LIN {X 0,Y 474.698,Z 275.654,A -85,B 0,C 180,E1 -7395.456,E2 -7395.456} C_VEL
LIN {X 0,Y 474.663,Z 275.673,A -85,B 0,C 180,E1 -7399.01,E2 -7399.01} C_VEL
LIN {X 0,Y 474.587,Z 275.663,A -85,B 0,C 180,E1 -7401.729,E2 -7401.729} C_VEL
LIN {X 0,Y 474.657,Z 275.67,A -85,B 0,C 180,E1 -7404.493,E2 -7404.493} C_VEL
LIN {X 0,Y 474.679,Z 275.656,A -85,B 0,C 180,E1 -7407.335,E2 -7407.335} C_VEL
LIN {X 0,Y 474.603,Z 275.676,A -85,B 0,C 180,E1 -7410.23,E2 -7410.23} C_VEL
LIN {X 0,Y 474.641,Z 275.673,A -85,B 0,C 180,E1 -7413.22,E2 -7413.22} C_VEL
LIN {X 0,Y 474.592,Z 275.678,A -85,B 0,C 180,E1 -7416.323,E2 -7416.323} C_VEL
LIN {X 0,Y 474.616,Z 275.673,A -85,B 0,C 180,E1 -7419.646,E2 -7419.646} C_VEL
LIN {X 0,Y 474.63,Z 275.671,A -85,B 0,C 180,E1 -7422.933,E2 -7422.933} C_VEL
LIN {X 0,Y 474.608,Z 275.668,A -85,B 0,C 180,E1 -7425.895,E2 -7425.895} C_VEL
LIN {X 0,Y 474.627,Z 275.678,A -85,B 0,C 180,E1 -7429.041,E2 -7429.041} C_VEL
LIN {X 0,Y 474.609,Z 275.671,A -85,B 0,C 180,E1 -7431.704,E2 -7431.704} C_VEL
LIN {X 0,Y 474.624,Z 275.678,A -85,B 0,C 180,E1 -7434.726,E2 -7434.726} C_VEL
LIN {X 0,Y 474.635,Z 275.669,A -85,B 0,C 180,E1 -7437.788,E2 -7437.788} C_VEL
LIN {X 0,Y 474.657,Z 275.717,A -85,B 0,C 180,E1 -7439.725,E2 -7439.725} C_VEL
LIN {X 0,Y 477.611,Z 285.664,A -85,B 0,C 180,E1 -7441.163,E2 -7441.163} C_VEL
LIN {X 0,Y 486.377,Z 304.406,A -85,B 0,C 180,E1 -7442.044,E2 -7442.044} C_VEL
LIN {X 0,Y 486.586,Z 308.524,A -85,B 0,C 180,E1 -7442.124,E2 -7442.124} C_VEL
LIN {X 0,Y 485.977,Z 352.152,A -85,B 0,C 180,E1 -7442.8,E2 -7442.8} C_VEL
LIN {X 0,Y 485.357,Z 358.003,A -85,B 0,C 180,E1 -7442.857,E2 -7442.857} C_VEL
LIN {X 0,Y 479.946,Z 377.102,A -85,B 0,C 180,E1 -7442.838,E2 -7442.838} C_VEL
LIN {X 0,Y 479.226,Z 382.961,A -85,B 0,C 180,E1 -7442.89,E2 -7442.89} C_VEL
LIN {X 0,Y 477.794,Z 488.089,A -85,B 0,C 180,E1 -7444.548,E2 -7444.548} C_VEL
LIN {X 0,Y 477.341,Z 503.327,A -85,B 0,C 180,E1 -7444.899,E2 -7444.899} C_VEL
LIN {X 0,Y 476.655,Z 519.69,A -85,B 0,C 180,E1 -7445.443,E2 -7445.443} C_VEL
LIN {X 0,Y 475.799,Z 535.126,A -85,B 0,C 180,E1 -7446.132,E2 -7446.132} C_VEL
LIN {X 0,Y 474.828,Z 550.129,A -85,B 0,C 180,E1 -7446.975,E2 -7446.975} C_VEL
LIN {X 0,Y 473.716,Z 565.062,A -85,B 0,C 180,E1 -7448,E2 -7448} C_VEL
LIN {X 0,Y 472.635,Z 578.371,A -85,B 0,C 180,E1 -7449.092,E2 -7449.092} C_VEL
LIN {X 0,Y 471.51,Z 591.755,A -85,B 0,C 180,E1 -7450.405,E2 -7450.405} C_VEL
LIN {X 0,Y 470.479,Z 603.142,A -85,B 0,C 180,E1 -7451.718,E2 -7451.718} C_VEL
LIN {X 0,Y 469.522,Z 615.062,A -85,B 0,C 180,E1 -7453.331,E2 -7453.331} C_VEL
LIN {X 0,Y 468.699,Z 625.549,A -85,B 0,C 180,E1 -7455.01,E2 -7455.01} C_VEL
LIN {X 0,Y 467.993,Z 634.788,A -85,B 0,C 180,E1 -7456.761,E2 -7456.761} C_VEL
LIN {X 0,Y 467.476,Z 643.328,A -85,B 0,C 180,E1 -7458.73,E2 -7458.73} C_VEL
LIN {X 0,Y 467.036,Z 650.904,A -85,B 0,C 180,E1 -7460.909,E2 -7460.909} C_VEL
LIN {X 0,Y 466.857,Z 655.603,A -85,B 0,C 180,E1 -7462.648,E2 -7462.648} C_VEL
LIN {X 0,Y 466.786,Z 658.459,A -85,B 0,C 180,E1 -7463.95,E2 -7463.95} C_VEL
LIN {X 0,Y 466.637,Z 661.374,A -85,B 0,C 180,E1 -7465.681,E2 -7465.681} C_VEL
LIN {X 0,Y 466.674,Z 663.284,A -85,B 0,C 180,E1 -7467.411,E2 -7467.411} C_VEL
LIN {X 0,Y 466.616,Z 664.26,A -85,B 0,C 180,E1 -7469.137,E2 -7469.137} C_VEL
LIN {X 0,Y 466.615,Z 664.276,A -85,B 0,C 180,E1 -7470.863,E2 -7470.863} C_VEL
LIN {X 0,Y 466.674,Z 663.368,A -85,B 0,C 180,E1 -7472.589,E2 -7472.589} C_VEL
LIN {X 0,Y 466.636,Z 661.491,A -85,B 0,C 180,E1 -7474.319,E2 -7474.319} C_VEL
LIN {X 0,Y 466.808,Z 657.814,A -85,B 0,C 180,E1 -7476.456,E2 -7476.456} C_VEL
LIN {X 0,Y 466.958,Z 653.633,A -85,B 0,C 180,E1 -7478.22,E2 -7478.22} C_VEL
LIN {X 0,Y 467.131,Z 648.378,A -85,B 0,C 180,E1 -7479.963,E2 -7479.963} C_VEL
LIN {X 0,Y 467.549,Z 641.906,A -85,B 0,C 180,E1 -7481.708,E2 -7481.708} C_VEL
LIN {X 0,Y 468.046,Z 634.141,A -85,B 0,C 180,E1 -7483.458,E2 -7483.458} C_VEL
LIN {X 0,Y 468.755,Z 624.825,A -85,B 0,C 180,E1 -7485.211,E2 -7485.211} C_VEL
LIN {X 0,Y 469.626,Z 613.968,A -85,B 0,C 180,E1 -7486.922,E2 -7486.922} C_VEL
LIN {X 0,Y 470.594,Z 602.088,A -85,B 0,C 180,E1 -7488.503,E2 -7488.503} C_VEL
LIN {X 0,Y 471.667,Z 589.425,A -85,B 0,C 180,E1 -7489.928,E2 -7489.928} C_VEL
LIN {X 0,Y 472.899,Z 575.579,A -85,B 0,C 180,E1 -7491.238,E2 -7491.238} C_VEL
LIN {X 0,Y 473.973,Z 561.898,A -85,B 0,C 180,E1 -7492.331,E2 -7492.331} C_VEL
LIN {X 0,Y 475.059,Z 546.493,A -85,B 0,C 180,E1 -7493.344,E2 -7493.344} C_VEL
LIN {X 0,Y 475.946,Z 531.63,A -85,B 0,C 180,E1 -7494.132,E2 -7494.132} C_VEL
LIN {X 0,Y 476.877,Z 515.29,A -85,B 0,C 180,E1 -7494.807,E2 -7494.807} C_VEL
LIN {X 0,Y 477.391,Z 500.575,A -85,B 0,C 180,E1 -7495.273,E2 -7495.273} C_VEL
LIN {X 0,Y 477.922,Z 482.833,A -85,B 0,C 180,E1 -7495.638,E2 -7495.638} C_VEL
LIN {X 0,Y 480.341,Z 306.951,A -85,B 0,C 180,E1 -7498.393,E2 -7498.393} C_VEL
LIN {X 0,Y 470.381,Z 285.74,A -85,B 0,C 180,E1 -7499.424,E2 -7499.424} C_VEL
LIN {X 0,Y 467.558,Z 276.56,A -85,B 0,C 180,E1 -7500.82,E2 -7500.82} C_VEL
LIN {X 0,Y 467.585,Z 276.553,A -85,B 0,C 180,E1 -7503.788,E2 -7503.788} C_VEL
LIN {X 0,Y 467.541,Z 276.547,A -85,B 0,C 180,E1 -7507.185,E2 -7507.185} C_VEL
LIN {X 0,Y 467.573,Z 276.551,A -85,B 0,C 180,E1 -7510.265,E2 -7510.265} C_VEL
LIN {X 0,Y 467.585,Z 276.548,A -85,B 0,C 180,E1 -7512.567,E2 -7512.567} C_VEL
LIN {X 0,Y 467.569,Z 276.553,A -85,B 0,C 180,E1 -7515.053,E2 -7515.053} C_VEL
LIN {X 0,Y 467.587,Z 276.553,A -85,B 0,C 180,E1 -7517.44,E2 -7517.44} C_VEL
LIN {X 0,Y 467.574,Z 276.554,A -85,B 0,C 180,E1 -7520.854,E2 -7520.854} C_VEL
LIN {X 0,Y 467.56,Z 276.552,A -85,B 0,C 180,E1 -7524.26,E2 -7524.26} C_VEL
LIN {X 0,Y 467.579,Z 276.547,A -85,B 0,C 180,E1 -7527.321,E2 -7527.321} C_VEL
LIN {X 0,Y 467.568,Z 276.554,A -85,B 0,C 180,E1 -7530.667,E2 -7530.667} C_VEL
LIN {X 0,Y 467.614,Z 276.543,A -85,B 0,C 180,E1 -7533.199,E2 -7533.199} C_VEL
LIN {X 0,Y 467.591,Z 276.548,A -85,B 0,C 180,E1 -7536.468,E2 -7536.468} C_VEL
LIN {X 0,Y 467.62,Z 276.545,A -85,B 0,C 180,E1 -7539.777,E2 -7539.777} C_VEL
LIN {X 0,Y 467.604,Z 276.547,A -85,B 0,C 180,E1 -7542.506,E2 -7542.506} C_VEL
LIN {X 0,Y 467.604,Z 276.544,A -85,B 0,C 180,E1 -7545.196,E2 -7545.196} C_VEL
LIN {X 0,Y 467.653,Z 276.54,A -85,B 0,C 180,E1 -7547.854,E2 -7547.854} C_VEL
LIN {X 0,Y 467.677,Z 276.534,A -85,B 0,C 180,E1 -7551.357,E2 -7551.357} C_VEL
LIN {X 0,Y 467.743,Z 276.53,A -85,B 0,C 180,E1 -7553.962,E2 -7553.962} C_VEL
LIN {X 0,Y 467.857,Z 276.506,A -85,B 0,C 180,E1 -7557.417,E2 -7557.417} C_VEL
LIN {X 0,Y 467.88,Z 276.512,A -85,B 0,C 180,E1 -7560,E2 -7560} C_VEL
LIN {X 0,Y 467.857,Z 276.516,A -85,B 0,C 180,E1 -7562.583,E2 -7562.583} C_VEL
LIN {X 0,Y 467.742,Z 276.527,A -85,B 0,C 180,E1 -7566.037,E2 -7566.037} C_VEL
LIN {X 0,Y 467.678,Z 276.542,A -85,B 0,C 180,E1 -7568.643,E2 -7568.643} C_VEL
LIN {X 0,Y 467.653,Z 276.537,A -85,B 0,C 180,E1 -7572.145,E2 -7572.145} C_VEL
LIN {X 0,Y 467.636,Z 276.543,A -85,B 0,C 180,E1 -7575.695,E2 -7575.695} C_VEL
LIN {X 0,Y 467.614,Z 276.549,A -85,B 0,C 180,E1 -7578.765,E2 -7578.765} C_VEL
LIN {X 0,Y 467.577,Z 276.553,A -85,B 0,C 180,E1 -7581.268,E2 -7581.268} C_VEL
LIN {X 0,Y 467.57,Z 276.552,A -85,B 0,C 180,E1 -7583.943,E2 -7583.943} C_VEL
LIN {X 0,Y 467.613,Z 276.553,A -85,B 0,C 180,E1 -7586.8,E2 -7586.8} C_VEL
LIN {X 0,Y 467.551,Z 276.555,A -85,B 0,C 180,E1 -7589.738,E2 -7589.738} C_VEL
LIN {X 0,Y 467.58,Z 276.557,A -85,B 0,C 180,E1 -7592.758,E2 -7592.758} C_VEL
LIN {X 0,Y 467.554,Z 276.554,A -85,B 0,C 180,E1 -7595.889,E2 -7595.889} C_VEL
LIN {X 0,Y 467.579,Z 276.557,A -85,B 0,C 180,E1 -7599.145,E2 -7599.145} C_VEL
LIN {X 0,Y 467.583,Z 276.558,A -85,B 0,C 180,E1 -7602.567,E2 -7602.567} C_VEL
LIN {X 0,Y 467.568,Z 276.559,A -85,B 0,C 180,E1 -7605.053,E2 -7605.053} C_VEL
LIN {X 0,Y 467.586,Z 276.553,A -85,B 0,C 180,E1 -7607.44,E2 -7607.44} C_VEL
LIN {X 0,Y 467.579,Z 276.557,A -85,B 0,C 180,E1 -7610.855,E2 -7610.855} C_VEL
LIN {X 0,Y 467.557,Z 276.559,A -85,B 0,C 180,E1 -7614.261,E2 -7614.261} C_VEL
LIN {X 0,Y 467.618,Z 276.563,A -85,B 0,C 180,E1 -7616.732,E2 -7616.732} C_VEL
LIN {X 0,Y 473.316,Z 295.045,A -85,B 0,C 180,E1 -7619.243,E2 -7619.243} C_VEL
LIN {X 0,Y 475.745,Z 303.396,A -85,B 0,C 180,E1 -7620.329,E2 -7620.329} C_VEL
LIN {X 0,Y 475.862,Z 305.952,A -85,B 0,C 180,E1 -7620.618,E2 -7620.618} C_VEL
LIN {X 0,Y 475.685,Z 309.709,A -85,B 0,C 180,E1 -7620.982,E2 -7620.982} C_VEL
LIN {X 0,Y 480.083,Z 335.198,A -85,B 0,C 180,E1 -7621.695,E2 -7621.695} C_VEL
LIN {X 0,Y 477.574,Z 515.045,A -85,B 0,C 180,E1 -7624.523,E2 -7624.523} C_VEL
LIN {X 0,Y 476.934,Z 530.938,A -85,B 0,C 180,E1 -7624.906,E2 -7624.906} C_VEL
LIN {X 0,Y 476.204,Z 547.344,A -85,B 0,C 180,E1 -7625.476,E2 -7625.476} C_VEL
LIN {X 0,Y 475.296,Z 561.77,A -85,B 0,C 180,E1 -7626.123,E2 -7626.123} C_VEL
LIN {X 0,Y 474.374,Z 576.069,A -85,B 0,C 180,E1 -7626.934,E2 -7626.934} C_VEL
LIN {X 0,Y 473.143,Z 591.267,A -85,B 0,C 180,E1 -7627.972,E2 -7627.972} C_VEL
LIN {X 0,Y 471.982,Z 605.787,A -85,B 0,C 180,E1 -7629.176,E2 -7629.176} C_VEL
LIN {X 0,Y 470.929,Z 618.532,A -85,B 0,C 180,E1 -7630.425,E2 -7630.425} C_VEL
LIN {X 0,Y 469.868,Z 631.368,A -85,B 0,C 180,E1 -7631.919,E2 -7631.919} C_VEL
LIN {X 0,Y 468.941,Z 643.342,A -85,B 0,C 180,E1 -7633.569,E2 -7633.569} C_VEL
LIN {X 0,Y 468.186,Z 653.464,A -85,B 0,C 180,E1 -7635.215,E2 -7635.215} C_VEL
LIN {X 0,Y 467.648,Z 662.611,A -85,B 0,C 180,E1 -7636.972,E2 -7636.972} C_VEL
LIN {X 0,Y 467.223,Z 670.275,A -85,B 0,C 180,E1 -7638.723,E2 -7638.723} C_VEL
LIN {X 0,Y 466.863,Z 677.966,A -85,B 0,C 180,E1 -7640.906,E2 -7640.906} C_VEL
LIN {X 0,Y 466.775,Z 682.744,A -85,B 0,C 180,E1 -7642.647,E2 -7642.647} C_VEL
LIN {X 0,Y 466.696,Z 685.653,A -85,B 0,C 180,E1 -7643.949,E2 -7643.949} C_VEL
LIN {X 0,Y 466.606,Z 688.604,A -85,B 0,C 180,E1 -7645.681,E2 -7645.681} C_VEL
LIN {X 0,Y 466.637,Z 690.549,A -85,B 0,C 180,E1 -7647.41,E2 -7647.41} C_VEL
LIN {X 0,Y 466.614,Z 691.513,A -85,B 0,C 180,E1 -7649.137,E2 -7649.137} C_VEL
LIN {X 0,Y 466.614,Z 691.512,A -85,B 0,C 180,E1 -7650.863,E2 -7650.863} C_VEL
LIN {X 0,Y 466.637,Z 690.548,A -85,B 0,C 180,E1 -7652.59,E2 -7652.59} C_VEL
LIN {X 0,Y 466.606,Z 688.603,A -85,B 0,C 180,E1 -7654.319,E2 -7654.319} C_VEL
LIN {X 0,Y 466.748,Z 684.941,A -85,B 0,C 180,E1 -7656.393,E2 -7656.393} C_VEL
LIN {X 0,Y 466.834,Z 680.493,A -85,B 0,C 180,E1 -7658.223,E2 -7658.223} C_VEL
LIN {X 0,Y 466.981,Z 675.097,A -85,B 0,C 180,E1 -7659.967,E2 -7659.967} C_VEL
LIN {X 0,Y 467.36,Z 668.451,A -85,B 0,C 180,E1 -7661.713,E2 -7661.713} C_VEL
LIN {X 0,Y 467.749,Z 660.487,A -85,B 0,C 180,E1 -7663.467,E2 -7663.467} C_VEL
LIN {X 0,Y 468.449,Z 650.979,A -85,B 0,C 180,E1 -7665.221,E2 -7665.221} C_VEL
LIN {X 0,Y 469.272,Z 639.594,A -85,B 0,C 180,E1 -7666.98,E2 -7666.98} C_VEL
LIN {X 0,Y 470.247,Z 627.776,A -85,B 0,C 180,E1 -7668.517,E2 -7668.517} C_VEL
LIN {X 0,Y 471.239,Z 615.474,A -85,B 0,C 180,E1 -7669.884,E2 -7669.884} C_VEL
LIN {X 0,Y 472.283,Z 602.081,A -85,B 0,C 180,E1 -7671.153,E2 -7671.153} C_VEL
LIN {X 0,Y 473.375,Z 588.383,A -85,B 0,C 180,E1 -7672.246,E2 -7672.246} C_VEL
LIN {X 0,Y 474.499,Z 573.377,A -85,B 0,C 180,E1 -7673.233,E2 -7673.233} C_VEL
LIN {X 0,Y 475.517,Z 558.339,A -85,B 0,C 180,E1 -7674.039,E2 -7674.039} C_VEL
LIN {X 0,Y 476.42,Z 542.396,A -85,B 0,C 180,E1 -7674.716,E2 -7674.716} C_VEL
LIN {X 0,Y 477.177,Z 526.233,A -85,B 0,C 180,E1 -7675.226,E2 -7675.226} C_VEL
LIN {X 0,Y 477.681,Z 509.478,A -85,B 0,C 180,E1 -7675.577,E2 -7675.577} C_VEL
LIN {X 0,Y 480.11,Z 334.584,A -85,B 0,C 180,E1 -7678.312,E2 -7678.312} C_VEL
LIN {X 0,Y 475.615,Z 309.029,A -85,B 0,C 180,E1 -7679.057,E2 -7679.057} C_VEL
LIN {X 0,Y 475.783,Z 303.384,A -85,B 0,C 180,E1 -7679.666,E2 -7679.666} C_VEL
LIN {X 0,Y 470.106,Z 284.516,A -85,B 0,C 180,E1 -7682.165,E2 -7682.165} C_VEL
LIN {X 0,Y 467.619,Z 276.543,A -85,B 0,C 180,E1 -7683.268,E2 -7683.268} C_VEL
LIN {X 0,Y 467.551,Z 276.558,A -85,B 0,C 180,E1 -7685.89,E2 -7685.89} C_VEL
LIN {X 0,Y 467.58,Z 276.555,A -85,B 0,C 180,E1 -7689.145,E2 -7689.145} C_VEL
LIN {X 0,Y 467.584,Z 276.551,A -85,B 0,C 180,E1 -7692.567,E2 -7692.567} C_VEL
LIN {X 0,Y 467.568,Z 276.554,A -85,B 0,C 180,E1 -7695.053,E2 -7695.053} C_VEL
LIN {X 0,Y 467.586,Z 276.551,A -85,B 0,C 180,E1 -7697.44,E2 -7697.44} C_VEL
LIN {X 0,Y 467.573,Z 276.55,A -85,B 0,C 180,E1 -7700.855,E2 -7700.855} C_VEL
LIN {X 0,Y 467.559,Z 276.551,A -85,B 0,C 180,E1 -7704.26,E2 -7704.26} C_VEL
LIN {X 0,Y 467.579,Z 276.553,A -85,B 0,C 180,E1 -7707.321,E2 -7707.321} C_VEL
LIN {X 0,Y 467.567,Z 276.551,A -85,B 0,C 180,E1 -7710.667,E2 -7710.667} C_VEL
LIN {X 0,Y 467.614,Z 276.55,A -85,B 0,C 180,E1 -7713.2,E2 -7713.2} C_VEL
LIN {X 0,Y 467.59,Z 276.549,A -85,B 0,C 180,E1 -7716.468,E2 -7716.468} C_VEL
LIN {X 0,Y 467.62,Z 276.532,A -85,B 0,C 180,E1 -7719.777,E2 -7719.777} C_VEL
LIN {X 0,Y 467.604,Z 276.547,A -85,B 0,C 180,E1 -7722.507,E2 -7722.507} C_VEL
LIN {X 0,Y 467.603,Z 276.541,A -85,B 0,C 180,E1 -7725.197,E2 -7725.197} C_VEL
LIN {X 0,Y 467.653,Z 276.536,A -85,B 0,C 180,E1 -7727.855,E2 -7727.855} C_VEL
LIN {X 0,Y 467.679,Z 276.536,A -85,B 0,C 180,E1 -7731.357,E2 -7731.357} C_VEL
LIN {X 0,Y 467.743,Z 276.516,A -85,B 0,C 180,E1 -7733.963,E2 -7733.963} C_VEL
LIN {X 0,Y 467.857,Z 276.518,A -85,B 0,C 180,E1 -7737.417,E2 -7737.417} C_VEL
LIN {X 0,Y 467.88,Z 276.501,A -85,B 0,C 180,E1 -7740,E2 -7740} C_VEL
LIN {X 0,Y 467.858,Z 276.509,A -85,B 0,C 180,E1 -7742.583,E2 -7742.583} C_VEL
LIN {X 0,Y 467.733,Z 276.528,A -85,B 0,C 180,E1 -7746.038,E2 -7746.038} C_VEL
LIN {X 0,Y 467.679,Z 276.523,A -85,B 0,C 180,E1 -7748.643,E2 -7748.643} C_VEL
LIN {X 0,Y 467.654,Z 276.541,A -85,B 0,C 180,E1 -7752.146,E2 -7752.146} C_VEL
LIN {X 0,Y 467.637,Z 276.533,A -85,B 0,C 180,E1 -7755.695,E2 -7755.695} C_VEL
LIN {X 0,Y 467.615,Z 276.551,A -85,B 0,C 180,E1 -7758.765,E2 -7758.765} C_VEL
LIN {X 0,Y 467.578,Z 276.539,A -85,B 0,C 180,E1 -7761.268,E2 -7761.268} C_VEL
LIN {X 0,Y 467.571,Z 276.55,A -85,B 0,C 180,E1 -7763.943,E2 -7763.943} C_VEL
LIN {X 0,Y 467.615,Z 276.543,A -85,B 0,C 180,E1 -7766.8,E2 -7766.8} C_VEL
LIN {X 0,Y 467.552,Z 276.553,A -85,B 0,C 180,E1 -7769.738,E2 -7769.738} C_VEL
LIN {X 0,Y 467.582,Z 276.553,A -85,B 0,C 180,E1 -7772.759,E2 -7772.759} C_VEL
LIN {X 0,Y 467.555,Z 276.552,A -85,B 0,C 180,E1 -7775.89,E2 -7775.89} C_VEL
LIN {X 0,Y 467.574,Z 276.551,A -85,B 0,C 180,E1 -7779.146,E2 -7779.146} C_VEL
LIN {X 0,Y 467.585,Z 276.545,A -85,B 0,C 180,E1 -7782.567,E2 -7782.567} C_VEL
LIN {X 0,Y 467.569,Z 276.55,A -85,B 0,C 180,E1 -7785.053,E2 -7785.053} C_VEL
LIN {X 0,Y 467.588,Z 276.552,A -85,B 0,C 180,E1 -7787.44,E2 -7787.44} C_VEL
LIN {X 0,Y 467.582,Z 276.554,A -85,B 0,C 180,E1 -7790.856,E2 -7790.856} C_VEL
LIN {X 0,Y 467.559,Z 276.552,A -85,B 0,C 180,E1 -7794.261,E2 -7794.261} C_VEL
LIN {X 0,Y 467.581,Z 276.542,A -85,B 0,C 180,E1 -7797.321,E2 -7797.321} C_VEL
LIN {X 0,Y 467.581,Z 276.568,A -85,B 0,C 180,E1 -7799.299,E2 -7799.299} C_VEL
LIN {X 0,Y 470.498,Z 286.066,A -85,B 0,C 180,E1 -7800.687,E2 -7800.687} C_VEL
LIN {X 0,Y 480.235,Z 306.732,A -85,B 0,C 180,E1 -7801.689,E2 -7801.689} C_VEL
LIN {X 0,Y 479.226,Z 382.961,A -85,B 0,C 180,E1 -7802.89,E2 -7802.89} C_VEL
LIN {X 0,Y 478.525,Z 388.81,A -85,B 0,C 180,E1 -7802.944,E2 -7802.944} C_VEL
LIN {X 0,Y 473.174,Z 407.9,A -85,B 0,C 180,E1 -7802.929,E2 -7802.929} C_VEL
LIN {X 0,Y 472.476,Z 413.75,A -85,B 0,C 180,E1 -7802.983,E2 -7802.983} C_VEL
LIN {X 0,Y 471.384,Z 488.455,A -85,B 0,C 180,E1 -7804.179,E2 -7804.179} C_VEL
LIN {X 0,Y 470.848,Z 505.377,A -85,B 0,C 180,E1 -7804.588,E2 -7804.588} C_VEL
LIN {X 0,Y 470.137,Z 521.212,A -85,B 0,C 180,E1 -7805.138,E2 -7805.138} C_VEL
LIN {X 0,Y 469.272,Z 536.355,A -85,B 0,C 180,E1 -7805.832,E2 -7805.832} C_VEL
LIN {X 0,Y 468.266,Z 550.66,A -85,B 0,C 180,E1 -7806.654,E2 -7806.654} C_VEL
LIN {X 0,Y 467.129,Z 565.276,A -85,B 0,C 180,E1 -7807.673,E2 -7807.673} C_VEL
LIN {X 0,Y 465.997,Z 578.584,A -85,B 0,C 180,E1 -7808.78,E2 -7808.78} C_VEL
LIN {X 0,Y 464.759,Z 591.969,A -85,B 0,C 180,E1 -7810.109,E2 -7810.109} C_VEL
LIN {X 0,Y 463.682,Z 603.355,A -85,B 0,C 180,E1 -7811.44,E2 -7811.44} C_VEL
LIN {X 0,Y 462.696,Z 614.91,A -85,B 0,C 180,E1 -7813.022,E2 -7813.022} C_VEL
LIN {X 0,Y 461.883,Z 624.527,A -85,B 0,C 180,E1 -7814.557,E2 -7814.557} C_VEL
LIN {X 0,Y 461.101,Z 633.901,A -85,B 0,C 180,E1 -7816.335,E2 -7816.335} C_VEL
LIN {X 0,Y 460.558,Z 641.75,A -85,B 0,C 180,E1 -7818.112,E2 -7818.112} C_VEL
LIN {X 0,Y 460.096,Z 648.3,A -85,B 0,C 180,E1 -7819.883,E2 -7819.883} C_VEL
LIN {X 0,Y 459.895,Z 653.592,A -85,B 0,C 180,E1 -7821.653,E2 -7821.653} C_VEL
LIN {X 0,Y 459.717,Z 658.082,A -85,B 0,C 180,E1 -7823.564,E2 -7823.564} C_VEL
LIN {X 0,Y 459.553,Z 661.583,A -85,B 0,C 180,E1 -7825.615,E2 -7825.615} C_VEL
LIN {X 0,Y 459.596,Z 663.492,A -85,B 0,C 180,E1 -7827.371,E2 -7827.371} C_VEL
LIN {X 0,Y 459.519,Z 664.467,A -85,B 0,C 180,E1 -7829.124,E2 -7829.124} C_VEL
LIN {X 0,Y 459.519,Z 664.483,A -85,B 0,C 180,E1 -7830.876,E2 -7830.876} C_VEL
LIN {X 0,Y 459.596,Z 663.574,A -85,B 0,C 180,E1 -7832.629,E2 -7832.629} C_VEL
LIN {X 0,Y 459.552,Z 661.698,A -85,B 0,C 180,E1 -7834.385,E2 -7834.385} C_VEL
LIN {X 0,Y 459.717,Z 658.262,A -85,B 0,C 180,E1 -7836.435,E2 -7836.435} C_VEL
LIN {X 0,Y 459.891,Z 653.839,A -85,B 0,C 180,E1 -7838.347,E2 -7838.347} C_VEL
LIN {X 0,Y 460.079,Z 648.585,A -85,B 0,C 180,E1 -7840.118,E2 -7840.118} C_VEL
LIN {X 0,Y 460.528,Z 642.113,A -85,B 0,C 180,E1 -7841.889,E2 -7841.889} C_VEL
LIN {X 0,Y 461.083,Z 634.348,A -85,B 0,C 180,E1 -7843.666,E2 -7843.666} C_VEL
LIN {X 0,Y 461.847,Z 625.032,A -85,B 0,C 180,E1 -7845.444,E2 -7845.444} C_VEL
LIN {X 0,Y 462.766,Z 614.174,A -85,B 0,C 180,E1 -7847.18,E2 -7847.18} C_VEL
LIN {X 0,Y 463.837,Z 602.292,A -85,B 0,C 180,E1 -7848.782,E2 -7848.782} C_VEL
LIN {X 0,Y 464.936,Z 589.63,A -85,B 0,C 180,E1 -7850.229,E2 -7850.229} C_VEL
LIN {X 0,Y 466.16,Z 577.067,A -85,B 0,C 180,E1 -7851.444,E2 -7851.444} C_VEL
LIN {X 0,Y 467.279,Z 563.561,A -85,B 0,C 180,E1 -7852.552,E2 -7852.552} C_VEL
LIN {X 0,Y 468.373,Z 549.154,A -85,B 0,C 180,E1 -7853.533,E2 -7853.533} C_VEL
LIN {X 0,Y 469.399,Z 532.954,A -85,B 0,C 180,E1 -7854.432,E2 -7854.432} C_VEL
LIN {X 0,Y 470.405,Z 516.245,A -85,B 0,C 180,E1 -7855.142,E2 -7855.142} C_VEL
LIN {X 0,Y 470.982,Z 500.763,A -85,B 0,C 180,E1 -7855.641,E2 -7855.641} C_VEL
LIN {X 0,Y 471.538,Z 483.554,A -85,B 0,C 180,E1 -7856.001,E2 -7856.001} C_VEL
LIN {X 0,Y 474.061,Z 308.964,A -85,B 0,C 180,E1 -7858.773,E2 -7858.773} C_VEL
LIN {X 0,Y 464.278,Z 288.306,A -85,B 0,C 180,E1 -7859.804,E2 -7859.804} C_VEL
LIN {X 0,Y 463.104,Z 285.806,A -85,B 0,C 180,E1 -7859.954,E2 -7859.954} C_VEL
LIN {X 0,Y 460.536,Z 277.44,A -85,B 0,C 180,E1 -7861.255,E2 -7861.255} C_VEL
LIN {X 0,Y 460.53,Z 277.435,A -85,B 0,C 180,E1 -7864.505,E2 -7864.505} C_VEL
LIN {X 0,Y 460.497,Z 277.43,A -85,B 0,C 180,E1 -7867.623,E2 -7867.623} C_VEL
LIN {X 0,Y 460.538,Z 277.427,A -85,B 0,C 180,E1 -7870.269,E2 -7870.269} C_VEL
LIN {X 0,Y 460.499,Z 277.436,A -85,B 0,C 180,E1 -7873.375,E2 -7873.375} C_VEL
LIN {X 0,Y 460.498,Z 277.432,A -85,B 0,C 180,E1 -7876.624,E2 -7876.624} C_VEL
LIN {X 0,Y 460.537,Z 277.429,A -85,B 0,C 180,E1 -7879.731,E2 -7879.731} C_VEL
LIN {X 0,Y 460.498,Z 277.431,A -85,B 0,C 180,E1 -7882.523,E2 -7882.523} C_VEL
LIN {X 0,Y 460.546,Z 277.428,A -85,B 0,C 180,E1 -7885.624,E2 -7885.624} C_VEL
LIN {X 0,Y 460.535,Z 277.426,A -85,B 0,C 180,E1 -7888.744,E2 -7888.744} C_VEL
LIN {X 0,Y 460.579,Z 277.412,A -85,B 0,C 180,E1 -7892.254,E2 -7892.254} C_VEL
LIN {X 0,Y 460.557,Z 277.427,A -85,B 0,C 180,E1 -7894.705,E2 -7894.705} C_VEL
LIN {X 0,Y 460.508,Z 277.421,A -85,B 0,C 180,E1 -7897.571,E2 -7897.571} C_VEL
LIN {X 0,Y 460.566,Z 277.424,A -85,B 0,C 180,E1 -7900.384,E2 -7900.384} C_VEL
LIN {X 0,Y 460.561,Z 277.416,A -85,B 0,C 180,E1 -7903.146,E2 -7903.146} C_VEL
LIN {X 0,Y 460.552,Z 277.424,A -85,B 0,C 180,E1 -7905.868,E2 -7905.868} C_VEL
LIN {X 0,Y 460.607,Z 277.42,A -85,B 0,C 180,E1 -7908.559,E2 -7908.559} C_VEL
LIN {X 0,Y 460.692,Z 277.404,A -85,B 0,C 180,E1 -7912.108,E2 -7912.108} C_VEL
LIN {X 0,Y 460.696,Z 277.412,A -85,B 0,C 180,E1 -7914.748,E2 -7914.748} C_VEL
LIN {X 0,Y 460.798,Z 277.385,A -85,B 0,C 180,E1 -7917.377,E2 -7917.377} C_VEL
LIN {X 0,Y 460.851,Z 277.388,A -85,B 0,C 180,E1 -7920,E2 -7920} C_VEL
LIN {X 0,Y 460.822,Z 277.391,A -85,B 0,C 180,E1 -7922.622,E2 -7922.622} C_VEL
LIN {X 0,Y 460.708,Z 277.404,A -85,B 0,C 180,E1 -7926.13,E2 -7926.13} C_VEL
LIN {X 0,Y 460.625,Z 277.418,A -85,B 0,C 180,E1 -7928.776,E2 -7928.776} C_VEL
LIN {X 0,Y 460.61,Z 277.416,A -85,B 0,C 180,E1 -7932.445,E2 -7932.445} C_VEL
LIN {X 0,Y 460.597,Z 277.419,A -85,B 0,C 180,E1 -7935.997,E2 -7935.997} C_VEL
LIN {X 0,Y 460.568,Z 277.428,A -85,B 0,C 180,E1 -7938.902,E2 -7938.902} C_VEL
LIN {X 0,Y 460.512,Z 277.432,A -85,B 0,C 180,E1 -7941.486,E2 -7941.486} C_VEL
LIN {X 0,Y 460.539,Z 277.43,A -85,B 0,C 180,E1 -7944.332,E2 -7944.332} C_VEL
LIN {X 0,Y 460.57,Z 277.428,A -85,B 0,C 180,E1 -7947.244,E2 -7947.244} C_VEL
LIN {X 0,Y 460.507,Z 277.434,A -85,B 0,C 180,E1 -7950.24,E2 -7950.24} C_VEL
LIN {X 0,Y 460.526,Z 277.434,A -85,B 0,C 180,E1 -7953.325,E2 -7953.325} C_VEL
LIN {X 0,Y 460.476,Z 277.441,A -85,B 0,C 180,E1 -7956.529,E2 -7956.529} C_VEL
LIN {X 0,Y 460.542,Z 277.436,A -85,B 0,C 180,E1 -7958.898,E2 -7958.898} C_VEL
LIN {X 0,Y 460.52,Z 277.435,A -85,B 0,C 180,E1 -7962.181,E2 -7962.181} C_VEL
LIN {X 0,Y 460.517,Z 277.434,A -85,B 0,C 180,E1 -7965.412,E2 -7965.412} C_VEL
LIN {X 0,Y 460.532,Z 277.434,A -85,B 0,C 180,E1 -7968.397,E2 -7968.397} C_VEL
LIN {X 0,Y 460.524,Z 277.433,A -85,B 0,C 180,E1 -7971.267,E2 -7971.267} C_VEL
LIN {X 0,Y 460.507,Z 277.43,A -85,B 0,C 180,E1 -7974.554,E2 -7974.554} C_VEL
LIN {X 0,Y 460.574,Z 277.577,A -85,B 0,C 180,E1 -7976.301,E2 -7976.301} C_VEL
LIN {X 0,Y 466.451,Z 296.278,A -85,B 0,C 180,E1 -7978.905,E2 -7978.905} C_VEL
LIN {X 0,Y 469.323,Z 306.823,A -85,B 0,C 180,E1 -7980.288,E2 -7980.288} C_VEL
LIN {X 0,Y 469.173,Z 309.378,A -85,B 0,C 180,E1 -7980.537,E2 -7980.537} C_VEL
LIN {X 0,Y 473.809,Z 335.907,A -85,B 0,C 180,E1 -7981.3,E2 -7981.3} C_VEL
LIN {X 0,Y 471.346,Z 505.455,A -85,B 0,C 180,E1 -7983.984,E2 -7983.984} C_VEL
LIN {X 0,Y 470.837,Z 522.804,A -85,B 0,C 180,E1 -7984.324,E2 -7984.324} C_VEL
LIN {X 0,Y 470.064,Z 539.941,A -85,B 0,C 180,E1 -7984.839,E2 -7984.839} C_VEL
LIN {X 0,Y 469.151,Z 555.906,A -85,B 0,C 180,E1 -7985.496,E2 -7985.496} C_VEL
LIN {X 0,Y 468.238,Z 569.698,A -85,B 0,C 180,E1 -7986.215,E2 -7986.215} C_VEL
LIN {X 0,Y 467.032,Z 585.074,A -85,B 0,C 180,E1 -7987.202,E2 -7987.202} C_VEL
LIN {X 0,Y 465.867,Z 599.292,A -85,B 0,C 180,E1 -7988.309,E2 -7988.309} C_VEL
LIN {X 0,Y 464.717,Z 612.527,A -85,B 0,C 180,E1 -7989.53,E2 -7989.53} C_VEL
LIN {X 0,Y 463.671,Z 623.84,A -85,B 0,C 180,E1 -7990.751,E2 -7990.751} C_VEL
LIN {X 0,Y 462.615,Z 636.173,A -85,B 0,C 180,E1 -7992.312,E2 -7992.312} C_VEL
LIN {X 0,Y 461.756,Z 646.509,A -85,B 0,C 180,E1 -7993.843,E2 -7993.843} C_VEL
LIN {X 0,Y 461.057,Z 655.739,A -85,B 0,C 180,E1 -7995.433,E2 -7995.433} C_VEL
LIN {X 0,Y 460.531,Z 664.437,A -85,B 0,C 180,E1 -7997.216,E2 -7997.216} C_VEL
LIN {X 0,Y 460.102,Z 671.717,A -85,B 0,C 180,E1 -7998.993,E2 -7998.993} C_VEL
LIN {X 0,Y 459.787,Z 677.758,A -85,B 0,C 180,E1 -8000.764,E2 -8000.764} C_VEL
LIN {X 0,Y 459.648,Z 683.613,A -85,B 0,C 180,E1 -8002.974,E2 -8002.974} C_VEL
LIN {X 0,Y 459.578,Z 687.037,A -85,B 0,C 180,E1 -8004.736,E2 -8004.736} C_VEL
LIN {X 0,Y 459.56,Z 689.527,A -85,B 0,C 180,E1 -8006.493,E2 -8006.493} C_VEL
LIN {X 0,Y 459.511,Z 690.931,A -85,B 0,C 180,E1 -8008.247,E2 -8008.247} C_VEL
LIN {X 0,Y 459.525,Z 691.46,A -85,B 0,C 180,E1 -8010,E2 -8010} C_VEL
LIN {X 0,Y 459.511,Z 690.93,A -85,B 0,C 180,E1 -8011.753,E2 -8011.753} C_VEL
LIN {X 0,Y 459.56,Z 689.525,A -85,B 0,C 180,E1 -8013.507,E2 -8013.507} C_VEL
LIN {X 0,Y 459.578,Z 687.037,A -85,B 0,C 180,E1 -8015.265,E2 -8015.265} C_VEL
LIN {X 0,Y 459.649,Z 683.616,A -85,B 0,C 180,E1 -8017.026,E2 -8017.026} C_VEL
LIN {X 0,Y 459.787,Z 677.76,A -85,B 0,C 180,E1 -8019.236,E2 -8019.236} C_VEL
LIN {X 0,Y 460.187,Z 670.065,A -85,B 0,C 180,E1 -8021.451,E2 -8021.451} C_VEL
LIN {X 0,Y 460.693,Z 661.381,A -85,B 0,C 180,E1 -8023.453,E2 -8023.453} C_VEL
LIN {X 0,Y 461.372,Z 652.012,A -85,B 0,C 180,E1 -8025.234,E2 -8025.234} C_VEL
LIN {X 0,Y 462.099,Z 642.375,A -85,B 0,C 180,E1 -8026.796,E2 -8026.796} C_VEL
LIN {X 0,Y 463.053,Z 631.15,A -85,B 0,C 180,E1 -8028.357,E2 -8028.357} C_VEL
LIN {X 0,Y 464.178,Z 618.702,A -85,B 0,C 180,E1 -8029.828,E2 -8029.828} C_VEL
LIN {X 0,Y 465.294,Z 605.565,A -85,B 0,C 180,E1 -8031.138,E2 -8031.138} C_VEL
LIN {X 0,Y 466.517,Z 591.038,A -85,B 0,C 180,E1 -8032.357,E2 -8032.357} C_VEL
LIN {X 0,Y 467.71,Z 576.615,A -85,B 0,C 180,E1 -8033.362,E2 -8033.362} C_VEL
LIN {X 0,Y 468.767,Z 561.519,A -85,B 0,C 180,E1 -8034.231,E2 -8034.231} C_VEL
LIN {X 0,Y 469.786,Z 545.793,A -85,B 0,C 180,E1 -8034.941,E2 -8034.941} C_VEL
LIN {X 0,Y 470.514,Z 529.754,A -85,B 0,C 180,E1 -8035.491,E2 -8035.491} C_VEL
LIN {X 0,Y 471.2,Z 512.491,A -85,B 0,C 180,E1 -8035.891,E2 -8035.891} C_VEL
LIN {X 0,Y 473.827,Z 335.539,A -85,B 0,C 180,E1 -8038.702,E2 -8038.702} C_VEL
LIN {X 0,Y 469.151,Z 308.918,A -85,B 0,C 180,E1 -8039.485,E2 -8039.485} C_VEL
LIN {X 0,Y 469.125,Z 305.443,A -85,B 0,C 180,E1 -8039.875,E2 -8039.875} C_VEL
LIN {X 0,Y 463.658,Z 287.149,A -85,B 0,C 180,E1 -8042.338,E2 -8042.338} C_VEL
LIN {X 0,Y 460.554,Z 277.424,A -85,B 0,C 180,E1 -8043.725,E2 -8043.725} C_VEL
LIN {X 0,Y 460.474,Z 277.438,A -85,B 0,C 180,E1 -8046.529,E2 -8046.529} C_VEL
LIN {X 0,Y 460.556,Z 277.429,A -85,B 0,C 180,E1 -8049.859,E2 -8049.859} C_VEL
LIN {X 0,Y 460.515,Z 277.433,A -85,B 0,C 180,E1 -8052.901,E2 -8052.901} C_VEL
LIN {X 0,Y 460.509,Z 277.43,A -85,B 0,C 180,E1 -8055.83,E2 -8055.83} C_VEL
LIN {X 0,Y 460.528,Z 277.429,A -85,B 0,C 180,E1 -8058.989,E2 -8058.989} C_VEL
LIN {X 0,Y 460.521,Z 277.433,A -85,B 0,C 180,E1 -8061.267,E2 -8061.267} C_VEL
LIN {X 0,Y 460.51,Z 277.43,A -85,B 0,C 180,E1 -8064.555,E2 -8064.555} C_VEL
LIN {X 0,Y 460.528,Z 277.43,A -85,B 0,C 180,E1 -8067.716,E2 -8067.716} C_VEL
LIN {X 0,Y 460.537,Z 277.428,A -85,B 0,C 180,E1 -8070.769,E2 -8070.769} C_VEL
LIN {X 0,Y 460.56,Z 277.427,A -85,B 0,C 180,E1 -8073.735,E2 -8073.735} C_VEL
LIN {X 0,Y 460.543,Z 277.428,A -85,B 0,C 180,E1 -8076.624,E2 -8076.624} C_VEL
LIN {X 0,Y 460.548,Z 277.414,A -85,B 0,C 180,E1 -8079.453,E2 -8079.453} C_VEL
LIN {X 0,Y 460.555,Z 277.424,A -85,B 0,C 180,E1 -8082.23,E2 -8082.23} C_VEL
LIN {X 0,Y 460.562,Z 277.422,A -85,B 0,C 180,E1 -8084.965,E2 -8084.965} C_VEL
LIN {X 0,Y 460.608,Z 277.415,A -85,B 0,C 180,E1 -8088.559,E2 -8088.559} C_VEL
LIN {X 0,Y 460.693,Z 277.401,A -85,B 0,C 180,E1 -8092.109,E2 -8092.109} C_VEL
LIN {X 0,Y 460.696,Z 277.397,A -85,B 0,C 180,E1 -8094.748,E2 -8094.748} C_VEL
LIN {X 0,Y 460.822,Z 277.395,A -85,B 0,C 180,E1 -8097.378,E2 -8097.378} C_VEL
LIN {X 0,Y 460.85,Z 277.376,A -85,B 0,C 180,E1 -8100,E2 -8100} C_VEL
LIN {X 0,Y 460.799,Z 277.389,A -85,B 0,C 180,E1 -8102.623,E2 -8102.623} C_VEL
LIN {X 0,Y 460.699,Z 277.404,A -85,B 0,C 180,E1 -8106.13,E2 -8106.13} C_VEL
LIN {X 0,Y 460.626,Z 277.402,A -85,B 0,C 180,E1 -8108.776,E2 -8108.776} C_VEL
LIN {X 0,Y 460.611,Z 277.42,A -85,B 0,C 180,E1 -8112.445,E2 -8112.445} C_VEL
LIN {X 0,Y 460.598,Z 277.408,A -85,B 0,C 180,E1 -8115.998,E2 -8115.998} C_VEL
LIN {X 0,Y 460.569,Z 277.431,A -85,B 0,C 180,E1 -8118.902,E2 -8118.902} C_VEL
LIN {X 0,Y 460.514,Z 277.416,A -85,B 0,C 180,E1 -8121.486,E2 -8121.486} C_VEL
LIN {X 0,Y 460.541,Z 277.427,A -85,B 0,C 180,E1 -8124.332,E2 -8124.332} C_VEL
LIN {X 0,Y 460.571,Z 277.413,A -85,B 0,C 180,E1 -8127.244,E2 -8127.244} C_VEL
LIN {X 0,Y 460.509,Z 277.431,A -85,B 0,C 180,E1 -8130.24,E2 -8130.24} C_VEL
LIN {X 0,Y 460.528,Z 277.431,A -85,B 0,C 180,E1 -8133.325,E2 -8133.325} C_VEL
LIN {X 0,Y 460.477,Z 277.438,A -85,B 0,C 180,E1 -8136.529,E2 -8136.529} C_VEL
LIN {X 0,Y 460.525,Z 277.428,A -85,B 0,C 180,E1 -8139.863,E2 -8139.863} C_VEL
LIN {X 0,Y 460.512,Z 277.428,A -85,B 0,C 180,E1 -8142.901,E2 -8142.901} C_VEL
LIN {X 0,Y 460.51,Z 277.424,A -85,B 0,C 180,E1 -8145.831,E2 -8145.831} C_VEL
LIN {X 0,Y 460.531,Z 277.435,A -85,B 0,C 180,E1 -8148.989,E2 -8148.989} C_VEL
LIN {X 0,Y 460.526,Z 277.427,A -85,B 0,C 180,E1 -8151.267,E2 -8151.267} C_VEL
LIN {X 0,Y 460.51,Z 277.433,A -85,B 0,C 180,E1 -8154.555,E2 -8154.555} C_VEL
LIN {X 0,Y 460.531,Z 277.423,A -85,B 0,C 180,E1 -8157.716,E2 -8157.716} C_VEL
LIN {X 0,Y 460.554,Z 277.522,A -85,B 0,C 180,E1 -8158.874,E2 -8158.874} C_VEL
LIN {X 0,Y 463.239,Z 286.303,A -85,B 0,C 180,E1 -8160.181,E2 -8160.181} C_VEL
LIN {X 0,Y 473.266,Z 307.258,A -85,B 0,C 180,E1 -8161.238,E2 -8161.238} C_VEL
LIN {X 0,Y 474.091,Z 308.97,A -85,B 0,C 180,E1 -8161.322,E2 -8161.322} C_VEL
LIN {X 0,Y 472.476,Z 413.75,A -85,B 0,C 180,E1 -8162.983,E2 -8162.983} C_VEL
LIN {X 0,Y 471.771,Z 419.6,A -85,B 0,C 180,E1 -8163.037,E2 -8163.037} C_VEL
LIN {X 0,Y 466.416,Z 438.687,A -85,B 0,C 180,E1 -8163.023,E2 -8163.023} C_VEL
LIN {X 0,Y 465.76,Z 444.534,A -85,B 0,C 180,E1 -8163.081,E2 -8163.081} C_VEL
LIN {X 0,Y 464.929,Z 491.789,A -85,B 0,C 180,E1 -8163.856,E2 -8163.856} C_VEL
LIN {X 0,Y 464.385,Z 507.426,A -85,B 0,C 180,E1 -8164.269,E2 -8164.269} C_VEL
LIN {X 0,Y 463.555,Z 524.02,A -85,B 0,C 180,E1 -8164.881,E2 -8164.881} C_VEL
LIN {X 0,Y 462.682,Z 538.073,A -85,B 0,C 180,E1 -8165.549,E2 -8165.549} C_VEL
LIN {X 0,Y 461.509,Z 553.85,A -85,B 0,C 180,E1 -8166.493,E2 -8166.493} C_VEL
LIN {X 0,Y 460.29,Z 568.329,A -85,B 0,C 180,E1 -8167.56,E2 -8167.56} C_VEL
LIN {X 0,Y 458.986,Z 582.301,A -85,B 0,C 180,E1 -8168.793,E2 -8168.793} C_VEL
LIN {X 0,Y 457.85,Z 594.207,A -85,B 0,C 180,E1 -8170.03,E2 -8170.03} C_VEL
LIN {X 0,Y 456.745,Z 605.336,A -85,B 0,C 180,E1 -8171.381,E2 -8171.381} C_VEL
LIN {X 0,Y 455.709,Z 616.529,A -85,B 0,C 180,E1 -8172.974,E2 -8172.974} C_VEL
LIN {X 0,Y 454.747,Z 627.194,A -85,B 0,C 180,E1 -8174.768,E2 -8174.768} C_VEL
LIN {X 0,Y 453.96,Z 636.217,A -85,B 0,C 180,E1 -8176.572,E2 -8176.572} C_VEL
LIN {X 0,Y 453.462,Z 643.75,A -85,B 0,C 180,E1 -8178.376,E2 -8178.376} C_VEL
LIN {X 0,Y 452.946,Z 651.324,A -85,B 0,C 180,E1 -8180.624,E2 -8180.624} C_VEL
LIN {X 0,Y 452.739,Z 656.022,A -85,B 0,C 180,E1 -8182.418,E2 -8182.418} C_VEL
LIN {X 0,Y 452.631,Z 658.877,A -85,B 0,C 180,E1 -8183.76,E2 -8183.76} C_VEL
LIN {X 0,Y 452.474,Z 661.791,A -85,B 0,C 180,E1 -8185.546,E2 -8185.546} C_VEL
LIN {X 0,Y 452.519,Z 663.699,A -85,B 0,C 180,E1 -8187.329,E2 -8187.329} C_VEL
LIN {X 0,Y 452.427,Z 664.674,A -85,B 0,C 180,E1 -8189.11,E2 -8189.11} C_VEL
LIN {X 0,Y 452.426,Z 664.69,A -85,B 0,C 180,E1 -8190.89,E2 -8190.89} C_VEL
LIN {X 0,Y 452.519,Z 663.781,A -85,B 0,C 180,E1 -8192.67,E2 -8192.67} C_VEL
LIN {X 0,Y 452.472,Z 661.905,A -85,B 0,C 180,E1 -8194.454,E2 -8194.454} C_VEL
LIN {X 0,Y 452.649,Z 658.658,A -85,B 0,C 180,E1 -8196.441,E2 -8196.441} C_VEL
LIN {X 0,Y 452.842,Z 654.046,A -85,B 0,C 180,E1 -8198.478,E2 -8198.478} C_VEL
LIN {X 0,Y 453.047,Z 648.792,A -85,B 0,C 180,E1 -8200.276,E2 -8200.276} C_VEL
LIN {X 0,Y 453.52,Z 642.321,A -85,B 0,C 180,E1 -8202.076,E2 -8202.076} C_VEL
LIN {X 0,Y 454.127,Z 634.555,A -85,B 0,C 180,E1 -8203.879,E2 -8203.879} C_VEL
LIN {X 0,Y 454.921,Z 625.239,A -85,B 0,C 180,E1 -8205.685,E2 -8205.685} C_VEL
LIN {X 0,Y 455.956,Z 614.086,A -85,B 0,C 180,E1 -8207.492,E2 -8207.492} C_VEL
LIN {X 0,Y 457.071,Z 602.497,A -85,B 0,C 180,E1 -8209.071,E2 -8209.071} C_VEL
LIN {X 0,Y 458.286,Z 589.602,A -85,B 0,C 180,E1 -8210.561,E2 -8210.561} C_VEL
LIN {X 0,Y 459.61,Z 575.986,A -85,B 0,C 180,E1 -8211.883,E2 -8211.883} C_VEL
LIN {X 0,Y 460.816,Z 562.302,A -85,B 0,C 180,E1 -8213.005,E2 -8213.005} C_VEL
LIN {X 0,Y 462.01,Z 546.986,A -85,B 0,C 180,E1 -8214.038,E2 -8214.038} C_VEL
LIN {X 0,Y 463.038,Z 532.026,A -85,B 0,C 180,E1 -8214.85,E2 -8214.85} C_VEL
LIN {X 0,Y 464.01,Z 515.68,A -85,B 0,C 180,E1 -8215.543,E2 -8215.543} C_VEL
LIN {X 0,Y 464.654,Z 499.904,A -85,B 0,C 180,E1 -8216.044,E2 -8216.044} C_VEL
LIN {X 0,Y 465.204,Z 482.777,A -85,B 0,C 180,E1 -8216.399,E2 -8216.399} C_VEL
LIN {X 0,Y 467.8,Z 311.03,A -85,B 0,C 180,E1 -8219.163,E2 -8219.163} C_VEL
LIN {X 0,Y 458.918,Z 292.227,A -85,B 0,C 180,E1 -8220.121,E2 -8220.121} C_VEL
LIN {X 0,Y 455.901,Z 286.089,A -85,B 0,C 180,E1 -8220.47,E2 -8220.47} C_VEL
LIN {X 0,Y 453.475,Z 278.311,A -85,B 0,C 180,E1 -8221.71,E2 -8221.71} C_VEL
LIN {X 0,Y 453.478,Z 278.312,A -85,B 0,C 180,E1 -8224.989,E2 -8224.989} C_VEL
LIN {X 0,Y 453.46,Z 278.311,A -85,B 0,C 180,E1 -8228.312,E2 -8228.312} C_VEL
LIN {X 0,Y 453.492,Z 278.306,A -85,B 0,C 180,E1 -8230.609,E2 -8230.609} C_VEL
LIN {X 0,Y 453.455,Z 278.312,A -85,B 0,C 180,E1 -8233.244,E2 -8233.244} C_VEL
LIN {X 0,Y 453.464,Z 278.307,A -85,B 0,C 180,E1 -8235.779,E2 -8235.779} C_VEL
LIN {X 0,Y 453.477,Z 278.306,A -85,B 0,C 180,E1 -8238.209,E2 -8238.209} C_VEL
LIN {X 0,Y 453.489,Z 278.308,A -85,B 0,C 180,E1 -8240.794,E2 -8240.794} C_VEL
LIN {X 0,Y 453.454,Z 278.31,A -85,B 0,C 180,E1 -8243.917,E2 -8243.917} C_VEL
LIN {X 0,Y 453.48,Z 278.302,A -85,B 0,C 180,E1 -8247.151,E2 -8247.151} C_VEL
LIN {X 0,Y 453.473,Z 278.308,A -85,B 0,C 180,E1 -8250.268,E2 -8250.268} C_VEL
LIN {X 0,Y 453.504,Z 278.301,A -85,B 0,C 180,E1 -8253.294,E2 -8253.294} C_VEL
LIN {X 0,Y 453.501,Z 278.303,A -85,B 0,C 180,E1 -8256.239,E2 -8256.239} C_VEL
LIN {X 0,Y 453.48,Z 278.302,A -85,B 0,C 180,E1 -8259.117,E2 -8259.117} C_VEL
LIN {X 0,Y 453.508,Z 278.301,A -85,B 0,C 180,E1 -8261.944,E2 -8261.944} C_VEL
LIN {X 0,Y 453.537,Z 278.288,A -85,B 0,C 180,E1 -8264.726,E2 -8264.726} C_VEL
LIN {X 0,Y 453.556,Z 278.297,A -85,B 0,C 180,E1 -8268.379,E2 -8268.379} C_VEL
LIN {X 0,Y 453.649,Z 278.281,A -85,B 0,C 180,E1 -8271.985,E2 -8271.985} C_VEL
LIN {X 0,Y 453.67,Z 278.287,A -85,B 0,C 180,E1 -8274.667,E2 -8274.667} C_VEL
LIN {X 0,Y 453.742,Z 278.263,A -85,B 0,C 180,E1 -8277.337,E2 -8277.337} C_VEL
LIN {X 0,Y 453.821,Z 278.264,A -85,B 0,C 180,E1 -8280,E2 -8280} C_VEL
LIN {X 0,Y 453.762,Z 278.269,A -85,B 0,C 180,E1 -8282.663,E2 -8282.663} C_VEL
LIN {X 0,Y 453.676,Z 278.28,A -85,B 0,C 180,E1 -8286.225,E2 -8286.225} C_VEL
LIN {X 0,Y 453.589,Z 278.291,A -85,B 0,C 180,E1 -8288.913,E2 -8288.913} C_VEL
LIN {X 0,Y 453.56,Z 278.294,A -85,B 0,C 180,E1 -8292.529,E2 -8292.529} C_VEL
LIN {X 0,Y 453.542,Z 278.299,A -85,B 0,C 180,E1 -8296.196,E2 -8296.196} C_VEL
LIN {X 0,Y 453.517,Z 278.308,A -85,B 0,C 180,E1 -8299.041,E2 -8299.041} C_VEL
LIN {X 0,Y 453.473,Z 278.307,A -85,B 0,C 180,E1 -8301.836,E2 -8301.836} C_VEL
LIN {X 0,Y 453.511,Z 278.307,A -85,B 0,C 180,E1 -8304.734,E2 -8304.734} C_VEL
LIN {X 0,Y 453.529,Z 278.302,A -85,B 0,C 180,E1 -8307.96,E2 -8307.96} C_VEL
LIN {X 0,Y 453.463,Z 278.313,A -85,B 0,C 180,E1 -8311.525,E2 -8311.525} C_VEL
LIN {X 0,Y 453.486,Z 278.314,A -85,B 0,C 180,E1 -8314.778,E2 -8314.778} C_VEL
LIN {X 0,Y 453.47,Z 278.314,A -85,B 0,C 180,E1 -8318.311,E2 -8318.311} C_VEL
LIN {X 0,Y 453.491,Z 278.314,A -85,B 0,C 180,E1 -8320.609,E2 -8320.609} C_VEL
LIN {X 0,Y 453.453,Z 278.316,A -85,B 0,C 180,E1 -8323.244,E2 -8323.244} C_VEL
LIN {X 0,Y 453.47,Z 278.311,A -85,B 0,C 180,E1 -8325.78,E2 -8325.78} C_VEL
LIN {X 0,Y 453.479,Z 278.312,A -85,B 0,C 180,E1 -8328.21,E2 -8328.21} C_VEL
LIN {X 0,Y 453.513,Z 278.309,A -85,B 0,C 180,E1 -8330.79,E2 -8330.79} C_VEL
LIN {X 0,Y 453.451,Z 278.315,A -85,B 0,C 180,E1 -8333.917,E2 -8333.917} C_VEL
LIN {X 0,Y 453.514,Z 278.345,A -85,B 0,C 180,E1 -8335.823,E2 -8335.823} C_VEL
LIN {X 0,Y 459.874,Z 298.534,A -85,B 0,C 180,E1 -8338.695,E2 -8338.695} C_VEL
LIN {X 0,Y 462.706,Z 308.908,A -85,B 0,C 180,E1 -8340.079,E2 -8340.079} C_VEL
LIN {X 0,Y 467.572,Z 336.764,A -85,B 0,C 180,E1 -8340.899,E2 -8340.899} C_VEL
LIN {X 0,Y 465.018,Z 502.944,A -85,B 0,C 180,E1 -8343.564,E2 -8343.564} C_VEL
LIN {X 0,Y 464.467,Z 521.656,A -85,B 0,C 180,E1 -8343.921,E2 -8343.921} C_VEL
LIN {X 0,Y 463.716,Z 538.213,A -85,B 0,C 180,E1 -8344.41,E2 -8344.41} C_VEL
LIN {X 0,Y 462.717,Z 554.57,A -85,B 0,C 180,E1 -8345.072,E2 -8345.072} C_VEL
LIN {X 0,Y 461.68,Z 569.904,A -85,B 0,C 180,E1 -8345.88,E2 -8345.88} C_VEL
LIN {X 0,Y 460.415,Z 584.867,A -85,B 0,C 180,E1 -8346.855,E2 -8346.855} C_VEL
LIN {X 0,Y 459.176,Z 599.085,A -85,B 0,C 180,E1 -8347.977,E2 -8347.977} C_VEL
LIN {X 0,Y 457.955,Z 612.318,A -85,B 0,C 180,E1 -8349.214,E2 -8349.214} C_VEL
LIN {X 0,Y 456.706,Z 625.569,A -85,B 0,C 180,E1 -8350.68,E2 -8350.68} C_VEL
LIN {X 0,Y 455.583,Z 637.602,A -85,B 0,C 180,E1 -8352.262,E2 -8352.262} C_VEL
LIN {X 0,Y 454.728,Z 647.847,A -85,B 0,C 180,E1 -8353.848,E2 -8353.848} C_VEL
LIN {X 0,Y 453.897,Z 657.815,A -85,B 0,C 180,E1 -8355.656,E2 -8355.656} C_VEL
LIN {X 0,Y 453.365,Z 666.205,A -85,B 0,C 180,E1 -8357.466,E2 -8357.466} C_VEL
LIN {X 0,Y 452.946,Z 673.135,A -85,B 0,C 180,E1 -8359.269,E2 -8359.269} C_VEL
LIN {X 0,Y 452.67,Z 678.815,A -85,B 0,C 180,E1 -8361.068,E2 -8361.068} C_VEL
LIN {X 0,Y 452.57,Z 683.405,A -85,B 0,C 180,E1 -8362.864,E2 -8362.864} C_VEL
LIN {X 0,Y 452.496,Z 686.83,A -85,B 0,C 180,E1 -8364.653,E2 -8364.653} C_VEL
LIN {X 0,Y 452.456,Z 689.319,A -85,B 0,C 180,E1 -8366.438,E2 -8366.438} C_VEL
LIN {X 0,Y 452.427,Z 690.724,A -85,B 0,C 180,E1 -8368.22,E2 -8368.22} C_VEL
LIN {X 0,Y 452.43,Z 691.253,A -85,B 0,C 180,E1 -8370,E2 -8370} C_VEL
LIN {X 0,Y 452.427,Z 690.723,A -85,B 0,C 180,E1 -8371.78,E2 -8371.78} C_VEL
LIN {X 0,Y 452.456,Z 689.317,A -85,B 0,C 180,E1 -8373.562,E2 -8373.562} C_VEL
LIN {X 0,Y 452.496,Z 686.829,A -85,B 0,C 180,E1 -8375.347,E2 -8375.347} C_VEL
LIN {X 0,Y 452.57,Z 683.407,A -85,B 0,C 180,E1 -8377.136,E2 -8377.136} C_VEL
LIN {X 0,Y 452.723,Z 677.551,A -85,B 0,C 180,E1 -8379.381,E2 -8379.381} C_VEL
LIN {X 0,Y 453.157,Z 669.855,A -85,B 0,C 180,E1 -8381.631,E2 -8381.631} C_VEL
LIN {X 0,Y 453.67,Z 661.169,A -85,B 0,C 180,E1 -8383.665,E2 -8383.665} C_VEL
LIN {X 0,Y 454.435,Z 651.801,A -85,B 0,C 180,E1 -8385.473,E2 -8385.473} C_VEL
LIN {X 0,Y 455.204,Z 642.163,A -85,B 0,C 180,E1 -8387.058,E2 -8387.058} C_VEL
LIN {X 0,Y 456.219,Z 630.938,A -85,B 0,C 180,E1 -8388.642,E2 -8388.642} C_VEL
LIN {X 0,Y 457.378,Z 618.883,A -85,B 0,C 180,E1 -8390.088,E2 -8390.088} C_VEL
LIN {X 0,Y 458.565,Z 605.352,A -85,B 0,C 180,E1 -8391.463,E2 -8391.463} C_VEL
LIN {X 0,Y 459.753,Z 592.258,A -85,B 0,C 180,E1 -8392.586,E2 -8392.586} C_VEL
LIN {X 0,Y 460.996,Z 578.419,A -85,B 0,C 180,E1 -8393.588,E2 -8393.588} C_VEL
LIN {X 0,Y 462.193,Z 562.396,A -85,B 0,C 180,E1 -8394.538,E2 -8394.538} C_VEL
LIN {X 0,Y 463.235,Z 546.881,A -85,B 0,C 180,E1 -8395.258,E2 -8395.258} C_VEL
LIN {X 0,Y 464.073,Z 530.456,A -85,B 0,C 180,E1 -8395.84,E2 -8395.84} C_VEL
LIN {X 0,Y 464.763,Z 513.987,A -85,B 0,C 180,E1 -8396.243,E2 -8396.243} C_VEL
LIN {X 0,Y 467.596,Z 337.685,A -85,B 0,C 180,E1 -8399.08,E2 -8399.08} C_VEL
LIN {X 0,Y 464.394,Z 318.567,A -85,B 0,C 180,E1 -8399.63,E2 -8399.63} C_VEL
LIN {X 0,Y 462.672,Z 308.749,A -85,B 0,C 180,E1 -8399.934,E2 -8399.934} C_VEL
LIN {X 0,Y 458.34,Z 293.454,A -85,B 0,C 180,E1 -8402.002,E2 -8402.002} C_VEL
LIN {X 0,Y 453.514,Z 278.306,A -85,B 0,C 180,E1 -8404.177,E2 -8404.177} C_VEL
LIN {X 0,Y 453.447,Z 278.314,A -85,B 0,C 180,E1 -8407.773,E2 -8407.773} C_VEL
LIN {X 0,Y 453.492,Z 278.309,A -85,B 0,C 180,E1 -8410.609,E2 -8410.609} C_VEL
LIN {X 0,Y 453.461,Z 278.314,A -85,B 0,C 180,E1 -8413.245,E2 -8413.245} C_VEL
LIN {X 0,Y 453.463,Z 278.308,A -85,B 0,C 180,E1 -8415.779,E2 -8415.779} C_VEL
LIN {X 0,Y 453.476,Z 278.303,A -85,B 0,C 180,E1 -8418.209,E2 -8418.209} C_VEL
LIN {X 0,Y 453.489,Z 278.304,A -85,B 0,C 180,E1 -8420.794,E2 -8420.794} C_VEL
LIN {X 0,Y 453.454,Z 278.309,A -85,B 0,C 180,E1 -8423.917,E2 -8423.917} C_VEL
LIN {X 0,Y 453.48,Z 278.309,A -85,B 0,C 180,E1 -8427.151,E2 -8427.151} C_VEL
LIN {X 0,Y 453.472,Z 278.305,A -85,B 0,C 180,E1 -8430.268,E2 -8430.268} C_VEL
LIN {X 0,Y 453.504,Z 278.308,A -85,B 0,C 180,E1 -8433.294,E2 -8433.294} C_VEL
LIN {X 0,Y 453.501,Z 278.303,A -85,B 0,C 180,E1 -8436.239,E2 -8436.239} C_VEL
LIN {X 0,Y 453.479,Z 278.298,A -85,B 0,C 180,E1 -8439.118,E2 -8439.118} C_VEL
LIN {X 0,Y 453.508,Z 278.302,A -85,B 0,C 180,E1 -8441.945,E2 -8441.945} C_VEL
LIN {X 0,Y 453.537,Z 278.301,A -85,B 0,C 180,E1 -8444.726,E2 -8444.726} C_VEL
LIN {X 0,Y 453.557,Z 278.292,A -85,B 0,C 180,E1 -8448.379,E2 -8448.379} C_VEL
LIN {X 0,Y 453.649,Z 278.279,A -85,B 0,C 180,E1 -8451.985,E2 -8451.985} C_VEL
LIN {X 0,Y 453.67,Z 278.271,A -85,B 0,C 180,E1 -8454.667,E2 -8454.667} C_VEL
LIN {X 0,Y 453.763,Z 278.275,A -85,B 0,C 180,E1 -8457.337,E2 -8457.337} C_VEL
LIN {X 0,Y 453.82,Z 278.251,A -85,B 0,C 180,E1 -8460,E2 -8460} C_VEL
LIN {X 0,Y 453.743,Z 278.268,A -85,B 0,C 180,E1 -8462.663,E2 -8462.663} C_VEL
LIN {X 0,Y 453.667,Z 278.28,A -85,B 0,C 180,E1 -8466.226,E2 -8466.226} C_VEL
LIN {X 0,Y 453.59,Z 278.279,A -85,B 0,C 180,E1 -8468.914,E2 -8468.914} C_VEL
LIN {X 0,Y 453.561,Z 278.299,A -85,B 0,C 180,E1 -8472.529,E2 -8472.529} C_VEL
LIN {X 0,Y 453.543,Z 278.287,A -85,B 0,C 180,E1 -8476.196,E2 -8476.196} C_VEL
LIN {X 0,Y 453.518,Z 278.306,A -85,B 0,C 180,E1 -8479.041,E2 -8479.041} C_VEL
LIN {X 0,Y 453.474,Z 278.291,A -85,B 0,C 180,E1 -8481.836,E2 -8481.836} C_VEL
LIN {X 0,Y 453.513,Z 278.307,A -85,B 0,C 180,E1 -8484.735,E2 -8484.735} C_VEL
LIN {X 0,Y 453.53,Z 278.286,A -85,B 0,C 180,E1 -8487.96,E2 -8487.96} C_VEL
LIN {X 0,Y 453.464,Z 278.307,A -85,B 0,C 180,E1 -8491.525,E2 -8491.525} C_VEL
LIN {X 0,Y 453.488,Z 278.308,A -85,B 0,C 180,E1 -8494.778,E2 -8494.778} C_VEL
LIN {X 0,Y 453.462,Z 278.299,A -85,B 0,C 180,E1 -8498.312,E2 -8498.312} C_VEL
LIN {X 0,Y 453.492,Z 278.309,A -85,B 0,C 180,E1 -8500.609,E2 -8500.609} C_VEL
LIN {X 0,Y 453.455,Z 278.311,A -85,B 0,C 180,E1 -8503.245,E2 -8503.245} C_VEL
LIN {X 0,Y 453.465,Z 278.302,A -85,B 0,C 180,E1 -8505.779,E2 -8505.779} C_VEL
LIN {X 0,Y 453.478,Z 278.31,A -85,B 0,C 180,E1 -8508.21,E2 -8508.21} C_VEL
LIN {X 0,Y 453.509,Z 278.307,A -85,B 0,C 180,E1 -8510.791,E2 -8510.791} C_VEL
LIN {X 0,Y 453.453,Z 278.304,A -85,B 0,C 180,E1 -8513.917,E2 -8513.917} C_VEL
LIN {X 0,Y 453.482,Z 278.295,A -85,B 0,C 180,E1 -8517.151,E2 -8517.151} C_VEL
LIN {X 0,Y 453.494,Z 278.369,A -85,B 0,C 180,E1 -8518.416,E2 -8518.416} C_VEL
LIN {X 0,Y 456.032,Z 286.421,A -85,B 0,C 180,E1 -8519.658,E2 -8519.658} C_VEL
LIN {X 0,Y 467.662,Z 310.68,A -85,B 0,C 180,E1 -8520.916,E2 -8520.916} C_VEL
LIN {X 0,Y 467.758,Z 318.24,A -85,B 0,C 180,E1 -8521.053,E2 -8521.053} C_VEL
LIN {X 0,Y 465.76,Z 444.534,A -85,B 0,C 180,E1 -8523.081,E2 -8523.081} C_VEL
LIN {X 0,Y 465.1,Z 450.389,A -85,B 0,C 180,E1 -8523.138,E2 -8523.138} C_VEL
LIN {X 0,Y 459.702,Z 469.494,A -85,B 0,C 180,E1 -8523.123,E2 -8523.123} C_VEL
LIN {X 0,Y 458.991,Z 475.352,A -85,B 0,C 180,E1 -8523.178,E2 -8523.178} C_VEL
LIN {X 0,Y 458.464,Z 495.531,A -85,B 0,C 180,E1 -8523.548,E2 -8523.548} C_VEL
LIN {X 0,Y 457.852,Z 511.257,A -85,B 0,C 180,E1 -8523.996,E2 -8523.996} C_VEL
LIN {X 0,Y 456.873,Z 528.125,A -85,B 0,C 180,E1 -8524.67,E2 -8524.67} C_VEL
LIN {X 0,Y 455.85,Z 543.098,A -85,B 0,C 180,E1 -8525.453,E2 -8525.453} C_VEL
LIN {X 0,Y 454.633,Z 558.131,A -85,B 0,C 180,E1 -8526.423,E2 -8526.423} C_VEL
LIN {X 0,Y 453.346,Z 572.622,A -85,B 0,C 180,E1 -8527.558,E2 -8527.558} C_VEL
LIN {X 0,Y 452.028,Z 586.229,A -85,B 0,C 180,E1 -8528.833,E2 -8528.833} C_VEL
LIN {X 0,Y 450.785,Z 598.293,A -85,B 0,C 180,E1 -8530.178,E2 -8530.178} C_VEL
LIN {X 0,Y 449.649,Z 608.904,A -85,B 0,C 180,E1 -8531.548,E2 -8531.548} C_VEL
LIN {X 0,Y 448.691,Z 618.523,A -85,B 0,C 180,E1 -8532.983,E2 -8532.983} C_VEL
LIN {X 0,Y 447.722,Z 628.626,A -85,B 0,C 180,E1 -8534.756,E2 -8534.756} C_VEL
LIN {X 0,Y 446.997,Z 636.428,A -85,B 0,C 180,E1 -8536.359,E2 -8536.359} C_VEL
LIN {X 0,Y 446.461,Z 643.96,A -85,B 0,C 180,E1 -8538.192,E2 -8538.192} C_VEL
LIN {X 0,Y 445.906,Z 651.534,A -85,B 0,C 180,E1 -8540.474,E2 -8540.474} C_VEL
LIN {X 0,Y 445.64,Z 657.284,A -85,B 0,C 180,E1 -8542.752,E2 -8542.752} C_VEL
LIN {X 0,Y 445.507,Z 660.654,A -85,B 0,C 180,E1 -8544.569,E2 -8544.569} C_VEL
LIN {X 0,Y 445.407,Z 663.104,A -85,B 0,C 180,E1 -8546.381,E2 -8546.381} C_VEL
LIN {X 0,Y 445.375,Z 664.499,A -85,B 0,C 180,E1 -8548.191,E2 -8548.191} C_VEL
LIN {X 0,Y 445.339,Z 665.038,A -85,B 0,C 180,E1 -8550,E2 -8550} C_VEL
LIN {X 0,Y 445.374,Z 664.547,A -85,B 0,C 180,E1 -8551.809,E2 -8551.809} C_VEL
LIN {X 0,Y 445.406,Z 663.2,A -85,B 0,C 180,E1 -8553.619,E2 -8553.619} C_VEL
LIN {X 0,Y 445.507,Z 660.799,A -85,B 0,C 180,E1 -8555.431,E2 -8555.431} C_VEL
LIN {X 0,Y 445.632,Z 657.487,A -85,B 0,C 180,E1 -8557.248,E2 -8557.248} C_VEL
LIN {X 0,Y 445.899,Z 651.798,A -85,B 0,C 180,E1 -8559.526,E2 -8559.526} C_VEL
LIN {X 0,Y 446.418,Z 644.311,A -85,B 0,C 180,E1 -8561.809,E2 -8561.809} C_VEL
LIN {X 0,Y 447.085,Z 635.825,A -85,B 0,C 180,E1 -8563.87,E2 -8563.87} C_VEL
LIN {X 0,Y 447.92,Z 626.666,A -85,B 0,C 180,E1 -8565.703,E2 -8565.703} C_VEL
LIN {X 0,Y 448.829,Z 617.238,A -85,B 0,C 180,E1 -8567.308,E2 -8567.308} C_VEL
LIN {X 0,Y 449.939,Z 606.242,A -85,B 0,C 180,E1 -8568.912,E2 -8568.912} C_VEL
LIN {X 0,Y 451.228,Z 593.616,A -85,B 0,C 180,E1 -8570.468,E2 -8570.468} C_VEL
LIN {X 0,Y 452.64,Z 579.917,A -85,B 0,C 180,E1 -8571.878,E2 -8571.878} C_VEL
LIN {X 0,Y 453.895,Z 566.804,A -85,B 0,C 180,E1 -8573.014,E2 -8573.014} C_VEL
LIN {X 0,Y 455.078,Z 553.543,A -85,B 0,C 180,E1 -8573.989,E2 -8573.989} C_VEL
LIN {X 0,Y 456.105,Z 539.82,A -85,B 0,C 180,E1 -8574.827,E2 -8574.827} C_VEL
LIN {X 0,Y 457.143,Z 524.93,A -85,B 0,C 180,E1 -8575.558,E2 -8575.558} C_VEL
LIN {X 0,Y 457.97,Z 508.615,A -85,B 0,C 180,E1 -8576.18,E2 -8576.18} C_VEL
LIN {X 0,Y 458.586,Z 494.01,A -85,B 0,C 180,E1 -8576.579,E2 -8576.579} C_VEL
LIN {X 0,Y 459.166,Z 462.89,A -85,B 0,C 180,E1 -8577.119,E2 -8577.119} C_VEL
LIN {X 0,Y 461.572,Z 312.915,A -85,B 0,C 180,E1 -8579.565,E2 -8579.565} C_VEL
LIN {X 0,Y 452.129,Z 293.234,A -85,B 0,C 180,E1 -8580.607,E2 -8580.607} C_VEL
LIN {X 0,Y 448.7,Z 286.461,A -85,B 0,C 180,E1 -8580.994,E2 -8580.994} C_VEL
LIN {X 0,Y 446.407,Z 279.184,A -85,B 0,C 180,E1 -8582.196,E2 -8582.196} C_VEL
LIN {X 0,Y 446.427,Z 279.189,A -85,B 0,C 180,E1 -8585.053,E2 -8585.053} C_VEL
LIN {X 0,Y 446.412,Z 279.19,A -85,B 0,C 180,E1 -8588.079,E2 -8588.079} C_VEL
LIN {X 0,Y 446.426,Z 279.189,A -85,B 0,C 180,E1 -8590.917,E2 -8590.917} C_VEL
LIN {X 0,Y 446.4,Z 279.192,A -85,B 0,C 180,E1 -8593.846,E2 -8593.846} C_VEL
LIN {X 0,Y 446.398,Z 279.187,A -85,B 0,C 180,E1 -8596.403,E2 -8596.403} C_VEL
LIN {X 0,Y 446.425,Z 279.183,A -85,B 0,C 180,E1 -8599.082,E2 -8599.082} C_VEL
LIN {X 0,Y 446.407,Z 279.185,A -85,B 0,C 180,E1 -8602.121,E2 -8602.121} C_VEL
LIN {X 0,Y 446.428,Z 279.188,A -85,B 0,C 180,E1 -8605.477,E2 -8605.477} C_VEL
LIN {X 0,Y 446.413,Z 279.184,A -85,B 0,C 180,E1 -8608.699,E2 -8608.699} C_VEL
LIN {X 0,Y 446.482,Z 279.169,A -85,B 0,C 180,E1 -8611.821,E2 -8611.821} C_VEL
LIN {X 0,Y 446.456,Z 279.185,A -85,B 0,C 180,E1 -8614.848,E2 -8614.848} C_VEL
LIN {X 0,Y 446.446,Z 279.17,A -85,B 0,C 180,E1 -8618.245,E2 -8618.245} C_VEL
LIN {X 0,Y 446.454,Z 279.181,A -85,B 0,C 180,E1 -8621.649,E2 -8621.649} C_VEL
LIN {X 0,Y 446.505,Z 279.161,A -85,B 0,C 180,E1 -8624.48,E2 -8624.48} C_VEL
LIN {X 0,Y 446.514,Z 279.174,A -85,B 0,C 180,E1 -8628.193,E2 -8628.193} C_VEL
LIN {X 0,Y 446.597,Z 279.159,A -85,B 0,C 180,E1 -8631.858,E2 -8631.858} C_VEL
LIN {X 0,Y 446.644,Z 279.161,A -85,B 0,C 180,E1 -8634.582,E2 -8634.582} C_VEL
LIN {X 0,Y 446.661,Z 279.145,A -85,B 0,C 180,E1 -8638.197,E2 -8638.197} C_VEL
LIN {X 0,Y 446.791,Z 279.14,A -85,B 0,C 180,E1 -8640,E2 -8640} C_VEL
LIN {X 0,Y 446.706,Z 279.146,A -85,B 0,C 180,E1 -8642.705,E2 -8642.705} C_VEL
LIN {X 0,Y 446.645,Z 279.156,A -85,B 0,C 180,E1 -8646.324,E2 -8646.324} C_VEL
LIN {X 0,Y 446.535,Z 279.167,A -85,B 0,C 180,E1 -8649.055,E2 -8649.055} C_VEL
LIN {X 0,Y 446.518,Z 279.174,A -85,B 0,C 180,E1 -8652.73,E2 -8652.73} C_VEL
LIN {X 0,Y 446.493,Z 279.177,A -85,B 0,C 180,E1 -8656.228,E2 -8656.228} C_VEL
LIN {X 0,Y 446.466,Z 279.185,A -85,B 0,C 180,E1 -8659.303,E2 -8659.303} C_VEL
LIN {X 0,Y 446.415,Z 279.188,A -85,B 0,C 180,E1 -8662.2,E2 -8662.2} C_VEL
LIN {X 0,Y 446.455,Z 279.189,A -85,B 0,C 180,E1 -8665.152,E2 -8665.152} C_VEL
LIN {X 0,Y 446.481,Z 279.181,A -85,B 0,C 180,E1 -8668.179,E2 -8668.179} C_VEL
LIN {X 0,Y 446.416,Z 279.191,A -85,B 0,C 180,E1 -8671.775,E2 -8671.775} C_VEL
LIN {X 0,Y 446.428,Z 279.193,A -85,B 0,C 180,E1 -8674.523,E2 -8674.523} C_VEL
LIN {X 0,Y 446.427,Z 279.19,A -85,B 0,C 180,E1 -8678.082,E2 -8678.082} C_VEL
LIN {X 0,Y 446.424,Z 279.194,A -85,B 0,C 180,E1 -8680.918,E2 -8680.918} C_VEL
LIN {X 0,Y 446.399,Z 279.193,A -85,B 0,C 180,E1 -8683.846,E2 -8683.846} C_VEL
LIN {X 0,Y 446.418,Z 279.193,A -85,B 0,C 180,E1 -8686.4,E2 -8686.4} C_VEL
LIN {X 0,Y 446.449,Z 279.186,A -85,B 0,C 180,E1 -8689.803,E2 -8689.803} C_VEL
LIN {X 0,Y 446.406,Z 279.192,A -85,B 0,C 180,E1 -8692.121,E2 -8692.121} C_VEL
LIN {X 0,Y 446.48,Z 279.268,A -85,B 0,C 180,E1 -8695.35,E2 -8695.35} C_VEL
LIN {X 0,Y 452.583,Z 298.299,A -85,B 0,C 180,E1 -8698.132,E2 -8698.132} C_VEL
LIN {X 0,Y 455.699,Z 308.967,A -85,B 0,C 180,E1 -8699.576,E2 -8699.576} C_VEL
LIN {X 0,Y 456.887,Z 312.062,A -85,B 0,C 180,E1 -8699.718,E2 -8699.718} C_VEL
LIN {X 0,Y 461.34,Z 337.604,A -85,B 0,C 180,E1 -8700.485,E2 -8700.485} C_VEL
LIN {X 0,Y 458.7,Z 502.318,A -85,B 0,C 180,E1 -8703.164,E2 -8703.164} C_VEL
LIN {X 0,Y 458.162,Z 520.594,A -85,B 0,C 180,E1 -8703.511,E2 -8703.511} C_VEL
LIN {X 0,Y 457.451,Z 535.721,A -85,B 0,C 180,E1 -8703.941,E2 -8703.941} C_VEL
LIN {X 0,Y 456.46,Z 551.952,A -85,B 0,C 180,E1 -8704.584,E2 -8704.584} C_VEL
LIN {X 0,Y 455.329,Z 567.228,A -85,B 0,C 180,E1 -8705.371,E2 -8705.371} C_VEL
LIN {X 0,Y 454,Z 583.074,A -85,B 0,C 180,E1 -8706.388,E2 -8706.388} C_VEL
LIN {X 0,Y 452.666,Z 597.581,A -85,B 0,C 180,E1 -8707.523,E2 -8707.523} C_VEL
LIN {X 0,Y 451.347,Z 611.035,A -85,B 0,C 180,E1 -8708.775,E2 -8708.775} C_VEL
LIN {X 0,Y 450.058,Z 623.422,A -85,B 0,C 180,E1 -8710.145,E2 -8710.145} C_VEL
LIN {X 0,Y 448.862,Z 635.754,A -85,B 0,C 180,E1 -8711.751,E2 -8711.751} C_VEL
LIN {X 0,Y 447.909,Z 645.851,A -85,B 0,C 180,E1 -8713.288,E2 -8713.288} C_VEL
LIN {X 0,Y 447.08,Z 655.319,A -85,B 0,C 180,E1 -8714.967,E2 -8714.967} C_VEL
LIN {X 0,Y 446.505,Z 664.019,A -85,B 0,C 180,E1 -8716.807,E2 -8716.807} C_VEL
LIN {X 0,Y 445.996,Z 671.299,A -85,B 0,C 180,E1 -8718.64,E2 -8718.64} C_VEL
LIN {X 0,Y 445.641,Z 677.34,A -85,B 0,C 180,E1 -8720.469,E2 -8720.469} C_VEL
LIN {X 0,Y 445.487,Z 683.197,A -85,B 0,C 180,E1 -8722.75,E2 -8722.75} C_VEL
LIN {X 0,Y 445.398,Z 686.622,A -85,B 0,C 180,E1 -8724.567,E2 -8724.567} C_VEL
LIN {X 0,Y 445.353,Z 689.112,A -85,B 0,C 180,E1 -8726.381,E2 -8726.381} C_VEL
LIN {X 0,Y 445.346,Z 690.517,A -85,B 0,C 180,E1 -8728.191,E2 -8728.191} C_VEL
LIN {X 0,Y 445.338,Z 691.046,A -85,B 0,C 180,E1 -8730,E2 -8730} C_VEL
LIN {X 0,Y 445.346,Z 690.516,A -85,B 0,C 180,E1 -8731.809,E2 -8731.809} C_VEL
LIN {X 0,Y 445.353,Z 689.109,A -85,B 0,C 180,E1 -8733.619,E2 -8733.619} C_VEL
LIN {X 0,Y 445.398,Z 686.621,A -85,B 0,C 180,E1 -8735.433,E2 -8735.433} C_VEL
LIN {X 0,Y 445.487,Z 683.198,A -85,B 0,C 180,E1 -8737.25,E2 -8737.25} C_VEL
LIN {X 0,Y 445.641,Z 677.34,A -85,B 0,C 180,E1 -8739.532,E2 -8739.532} C_VEL
LIN {X 0,Y 446.137,Z 669.645,A -85,B 0,C 180,E1 -8741.817,E2 -8741.817} C_VEL
LIN {X 0,Y 446.659,Z 660.957,A -85,B 0,C 180,E1 -8743.884,E2 -8743.884} C_VEL
LIN {X 0,Y 447.508,Z 651.589,A -85,B 0,C 180,E1 -8745.718,E2 -8745.718} C_VEL
LIN {X 0,Y 448.309,Z 641.95,A -85,B 0,C 180,E1 -8747.329,E2 -8747.329} C_VEL
LIN {X 0,Y 449.404,Z 630.726,A -85,B 0,C 180,E1 -8748.935,E2 -8748.935} C_VEL
LIN {X 0,Y 450.575,Z 619.073,A -85,B 0,C 180,E1 -8750.356,E2 -8750.356} C_VEL
LIN {X 0,Y 451.777,Z 606.319,A -85,B 0,C 180,E1 -8751.682,E2 -8751.682} C_VEL
LIN {X 0,Y 453.11,Z 592.044,A -85,B 0,C 180,E1 -8752.936,E2 -8752.936} C_VEL
LIN {X 0,Y 454.487,Z 577.679,A -85,B 0,C 180,E1 -8753.983,E2 -8753.983} C_VEL
LIN {X 0,Y 455.707,Z 562.182,A -85,B 0,C 180,E1 -8754.911,E2 -8754.911} C_VEL
LIN {X 0,Y 456.809,Z 546.667,A -85,B 0,C 180,E1 -8755.639,E2 -8755.639} C_VEL
LIN {X 0,Y 457.69,Z 530.24,A -85,B 0,C 180,E1 -8756.228,E2 -8756.228} C_VEL
LIN {X 0,Y 458.395,Z 514.14,A -85,B 0,C 180,E1 -8756.628,E2 -8756.628} C_VEL
LIN {X 0,Y 461.374,Z 338.588,A -85,B 0,C 180,E1 -8759.491,E2 -8759.491} C_VEL
LIN {X 0,Y 456.734,Z 311.329,A -85,B 0,C 180,E1 -8760.301,E2 -8760.301} C_VEL
LIN {X 0,Y 455.482,Z 308.399,A -85,B 0,C 180,E1 -8760.469,E2 -8760.469} C_VEL
LIN {X 0,Y 450.809,Z 292.679,A -85,B 0,C 180,E1 -8762.665,E2 -8762.665} C_VEL
LIN {X 0,Y 446.462,Z 279.187,A -85,B 0,C 180,E1 -8764.685,E2 -8764.685} C_VEL
LIN {X 0,Y 446.413,Z 279.191,A -85,B 0,C 180,E1 -8768.079,E2 -8768.079} C_VEL
LIN {X 0,Y 446.426,Z 279.189,A -85,B 0,C 180,E1 -8770.918,E2 -8770.918} C_VEL
LIN {X 0,Y 446.421,Z 279.186,A -85,B 0,C 180,E1 -8773.843,E2 -8773.843} C_VEL
LIN {X 0,Y 446.397,Z 279.186,A -85,B 0,C 180,E1 -8776.403,E2 -8776.403} C_VEL
LIN {X 0,Y 446.424,Z 279.187,A -85,B 0,C 180,E1 -8779.082,E2 -8779.082} C_VEL
LIN {X 0,Y 446.406,Z 279.185,A -85,B 0,C 180,E1 -8782.121,E2 -8782.121} C_VEL
LIN {X 0,Y 446.428,Z 279.188,A -85,B 0,C 180,E1 -8785.477,E2 -8785.477} C_VEL
LIN {X 0,Y 446.413,Z 279.188,A -85,B 0,C 180,E1 -8788.7,E2 -8788.7} C_VEL
LIN {X 0,Y 446.482,Z 279.179,A -85,B 0,C 180,E1 -8791.821,E2 -8791.821} C_VEL
LIN {X 0,Y 446.455,Z 279.186,A -85,B 0,C 180,E1 -8794.848,E2 -8794.848} C_VEL
LIN {X 0,Y 446.445,Z 279.181,A -85,B 0,C 180,E1 -8798.245,E2 -8798.245} C_VEL
LIN {X 0,Y 446.454,Z 279.182,A -85,B 0,C 180,E1 -8801.649,E2 -8801.649} C_VEL
LIN {X 0,Y 446.505,Z 279.175,A -85,B 0,C 180,E1 -8804.48,E2 -8804.48} C_VEL
LIN {X 0,Y 446.515,Z 279.169,A -85,B 0,C 180,E1 -8808.193,E2 -8808.193} C_VEL
LIN {X 0,Y 446.598,Z 279.157,A -85,B 0,C 180,E1 -8811.858,E2 -8811.858} C_VEL
LIN {X 0,Y 446.644,Z 279.145,A -85,B 0,C 180,E1 -8814.583,E2 -8814.583} C_VEL
LIN {X 0,Y 446.706,Z 279.154,A -85,B 0,C 180,E1 -8817.295,E2 -8817.295} C_VEL
LIN {X 0,Y 446.79,Z 279.127,A -85,B 0,C 180,E1 -8820,E2 -8820} C_VEL
LIN {X 0,Y 446.69,Z 279.147,A -85,B 0,C 180,E1 -8822.706,E2 -8822.706} C_VEL
LIN {X 0,Y 446.637,Z 279.157,A -85,B 0,C 180,E1 -8826.324,E2 -8826.324} C_VEL
LIN {X 0,Y 446.536,Z 279.159,A -85,B 0,C 180,E1 -8829.056,E2 -8829.056} C_VEL
LIN {X 0,Y 446.519,Z 279.179,A -85,B 0,C 180,E1 -8832.73,E2 -8832.73} C_VEL
LIN {X 0,Y 446.494,Z 279.165,A -85,B 0,C 180,E1 -8836.228,E2 -8836.228} C_VEL
LIN {X 0,Y 446.467,Z 279.181,A -85,B 0,C 180,E1 -8839.303,E2 -8839.303} C_VEL
LIN {X 0,Y 446.416,Z 279.17,A -85,B 0,C 180,E1 -8842.2,E2 -8842.2} C_VEL
LIN {X 0,Y 446.456,Z 279.185,A -85,B 0,C 180,E1 -8845.152,E2 -8845.152} C_VEL
LIN {X 0,Y 446.483,Z 279.164,A -85,B 0,C 180,E1 -8848.179,E2 -8848.179} C_VEL
LIN {X 0,Y 446.417,Z 279.184,A -85,B 0,C 180,E1 -8851.775,E2 -8851.775} C_VEL
LIN {X 0,Y 446.429,Z 279.187,A -85,B 0,C 180,E1 -8854.523,E2 -8854.523} C_VEL
LIN {X 0,Y 446.414,Z 279.176,A -85,B 0,C 180,E1 -8858.079,E2 -8858.079} C_VEL
LIN {X 0,Y 446.425,Z 279.185,A -85,B 0,C 180,E1 -8860.918,E2 -8860.918} C_VEL
LIN {X 0,Y 446.401,Z 279.189,A -85,B 0,C 180,E1 -8863.846,E2 -8863.846} C_VEL
LIN {X 0,Y 446.399,Z 279.184,A -85,B 0,C 180,E1 -8866.404,E2 -8866.404} C_VEL
LIN {X 0,Y 446.427,Z 279.19,A -85,B 0,C 180,E1 -8869.083,E2 -8869.083} C_VEL
LIN {X 0,Y 446.415,Z 279.178,A -85,B 0,C 180,E1 -8871.921,E2 -8871.921} C_VEL
LIN {X 0,Y 446.429,Z 279.187,A -85,B 0,C 180,E1 -8875.477,E2 -8875.477} C_VEL
LIN {X 0,Y 446.44,Z 279.296,A -85,B 0,C 180,E1 -8877.953,E2 -8877.953} C_VEL
LIN {X 0,Y 448.82,Z 286.697,A -85,B 0,C 180,E1 -8879.118,E2 -8879.118} C_VEL
LIN {X 0,Y 460.609,Z 310.849,A -85,B 0,C 180,E1 -8880.425,E2 -8880.425} C_VEL
LIN {X 0,Y 461.573,Z 313.01,A -85,B 0,C 180,E1 -8880.531,E2 -8880.531} C_VEL
LIN {X 0,Y 458.991,Z 475.352,A -85,B 0,C 180,E1 -8883.178,E2 -8883.178} C_VEL
LIN {X 0,Y 458.29,Z 479.284,A -85,B 0,C 180,E1 -8883.2,E2 -8883.2} C_VEL
LIN {X 0,Y 452.839,Z 491.631,A -85,B 0,C 180,E1 -8883.088,E2 -8883.088} C_VEL
LIN {X 0,Y 452.144,Z 495.519,A -85,B 0,C 180,E1 -8883.143,E2 -8883.143} C_VEL
LIN {X 0,Y 451.477,Z 511.477,A -85,B 0,C 180,E1 -8883.601,E2 -8883.601} C_VEL
LIN {X 0,Y 450.486,Z 528.342,A -85,B 0,C 180,E1 -8884.285,E2 -8884.285} C_VEL
LIN {X 0,Y 449.338,Z 544.005,A -85,B 0,C 180,E1 -8885.117,E2 -8885.117} C_VEL
LIN {X 0,Y 448.12,Z 558.345,A -85,B 0,C 180,E1 -8886.059,E2 -8886.059} C_VEL
LIN {X 0,Y 446.909,Z 571.549,A -85,B 0,C 180,E1 -8887.095,E2 -8887.095} C_VEL
LIN {X 0,Y 445.477,Z 585.406,A -85,B 0,C 180,E1 -8888.397,E2 -8888.397} C_VEL
LIN {X 0,Y 444.223,Z 596.57,A -85,B 0,C 180,E1 -8889.632,E2 -8889.632} C_VEL
LIN {X 0,Y 443.035,Z 607.501,A -85,B 0,C 180,E1 -8891.023,E2 -8891.023} C_VEL
LIN {X 0,Y 441.783,Z 619.28,A -85,B 0,C 180,E1 -8892.797,E2 -8892.797} C_VEL
LIN {X 0,Y 440.812,Z 628.837,A -85,B 0,C 180,E1 -8894.511,E2 -8894.511} C_VEL
LIN {X 0,Y 440.052,Z 636.639,A -85,B 0,C 180,E1 -8896.139,E2 -8896.139} C_VEL
LIN {X 0,Y 439.444,Z 644.172,A -85,B 0,C 180,E1 -8898,E2 -8898} C_VEL
LIN {X 0,Y 438.85,Z 651.745,A -85,B 0,C 180,E1 -8900.32,E2 -8900.32} C_VEL
LIN {X 0,Y 438.578,Z 657.493,A -85,B 0,C 180,E1 -8902.635,E2 -8902.635} C_VEL
LIN {X 0,Y 438.429,Z 660.863,A -85,B 0,C 180,E1 -8904.481,E2 -8904.481} C_VEL
LIN {X 0,Y 438.31,Z 663.313,A -85,B 0,C 180,E1 -8906.323,E2 -8906.323} C_VEL
LIN {X 0,Y 438.296,Z 664.706,A -85,B 0,C 180,E1 -8908.162,E2 -8908.162} C_VEL
LIN {X 0,Y 438.25,Z 665.245,A -85,B 0,C 180,E1 -8910,E2 -8910} C_VEL
LIN {X 0,Y 438.295,Z 664.754,A -85,B 0,C 180,E1 -8911.838,E2 -8911.838} C_VEL
LIN {X 0,Y 438.309,Z 663.407,A -85,B 0,C 180,E1 -8913.677,E2 -8913.677} C_VEL
LIN {X 0,Y 438.428,Z 661.005,A -85,B 0,C 180,E1 -8915.519,E2 -8915.519} C_VEL
LIN {X 0,Y 438.569,Z 657.694,A -85,B 0,C 180,E1 -8917.365,E2 -8917.365} C_VEL
LIN {X 0,Y 438.841,Z 652.005,A -85,B 0,C 180,E1 -8919.681,E2 -8919.681} C_VEL
LIN {X 0,Y 439.413,Z 644.518,A -85,B 0,C 180,E1 -8922,E2 -8922} C_VEL
LIN {X 0,Y 440.121,Z 636.033,A -85,B 0,C 180,E1 -8924.094,E2 -8924.094} C_VEL
LIN {X 0,Y 441.017,Z 626.873,A -85,B 0,C 180,E1 -8925.956,E2 -8925.956} C_VEL
LIN {X 0,Y 441.994,Z 617.444,A -85,B 0,C 180,E1 -8927.584,E2 -8927.584} C_VEL
LIN {X 0,Y 443.176,Z 606.447,A -85,B 0,C 180,E1 -8929.211,E2 -8929.211} C_VEL
LIN {X 0,Y 444.487,Z 594.096,A -85,B 0,C 180,E1 -8930.758,E2 -8930.758} C_VEL
LIN {X 0,Y 445.874,Z 581.404,A -85,B 0,C 180,E1 -8932.094,E2 -8932.094} C_VEL
LIN {X 0,Y 447.325,Z 567.007,A -85,B 0,C 180,E1 -8933.372,E2 -8933.372} C_VEL
LIN {X 0,Y 448.675,Z 552.157,A -85,B 0,C 180,E1 -8934.465,E2 -8934.465} C_VEL
LIN {X 0,Y 449.814,Z 538.028,A -85,B 0,C 180,E1 -8935.322,E2 -8935.322} C_VEL
LIN {X 0,Y 450.923,Z 522.533,A -85,B 0,C 180,E1 -8936.061,E2 -8936.061} C_VEL
LIN {X 0,Y 451.659,Z 506.981,A -85,B 0,C 180,E1 -8936.637,E2 -8936.637} C_VEL
LIN {X 0,Y 452.342,Z 490.946,A -85,B 0,C 180,E1 -8937.051,E2 -8937.051} C_VEL
LIN {X 0,Y 455.452,Z 315.192,A -85,B 0,C 180,E1 -8939.965,E2 -8939.965} C_VEL
LIN {X 0,Y 446.408,Z 296.353,A -85,B 0,C 180,E1 -8940.988,E2 -8940.988} C_VEL
LIN {X 0,Y 441.376,Z 286.517,A -85,B 0,C 180,E1 -8941.592,E2 -8941.592} C_VEL
LIN {X 0,Y 439.368,Z 280.057,A -85,B 0,C 180,E1 -8942.673,E2 -8942.673} C_VEL
LIN {X 0,Y 439.392,Z 280.059,A -85,B 0,C 180,E1 -8945.34,E2 -8945.34} C_VEL
LIN {X 0,Y 439.375,Z 280.067,A -85,B 0,C 180,E1 -8948.595,E2 -8948.595} C_VEL
LIN {X 0,Y 439.387,Z 280.068,A -85,B 0,C 180,E1 -8951.256,E2 -8951.256} C_VEL
LIN {X 0,Y 439.4,Z 280.064,A -85,B 0,C 180,E1 -8954.729,E2 -8954.729} C_VEL
LIN {X 0,Y 439.394,Z 280.062,A -85,B 0,C 180,E1 -8957.795,E2 -8957.795} C_VEL
LIN {X 0,Y 439.409,Z 280.059,A -85,B 0,C 180,E1 -8960.225,E2 -8960.225} C_VEL
LIN {X 0,Y 439.373,Z 280.064,A -85,B 0,C 180,E1 -8963.713,E2 -8963.713} C_VEL
LIN {X 0,Y 439.37,Z 280.059,A -85,B 0,C 180,E1 -8967.054,E2 -8967.054} C_VEL
LIN {X 0,Y 439.38,Z 280.064,A -85,B 0,C 180,E1 -8970.274,E2 -8970.274} C_VEL
LIN {X 0,Y 439.426,Z 280.055,A -85,B 0,C 180,E1 -8973.396,E2 -8973.396} C_VEL
LIN {X 0,Y 439.385,Z 280.062,A -85,B 0,C 180,E1 -8976.429,E2 -8976.429} C_VEL
LIN {X 0,Y 439.386,Z 280.062,A -85,B 0,C 180,E1 -8979.397,E2 -8979.397} C_VEL
LIN {X 0,Y 439.428,Z 280.055,A -85,B 0,C 180,E1 -8982.309,E2 -8982.309} C_VEL
LIN {X 0,Y 439.445,Z 280.048,A -85,B 0,C 180,E1 -8985.174,E2 -8985.174} C_VEL
LIN {X 0,Y 439.48,Z 280.05,A -85,B 0,C 180,E1 -8988.001,E2 -8988.001} C_VEL
LIN {X 0,Y 439.545,Z 280.038,A -85,B 0,C 180,E1 -8991.726,E2 -8991.726} C_VEL
LIN {X 0,Y 439.62,Z 280.035,A -85,B 0,C 180,E1 -8994.496,E2 -8994.496} C_VEL
LIN {X 0,Y 439.631,Z 280.021,A -85,B 0,C 180,E1 -8998.168,E2 -8998.168} C_VEL
LIN {X 0,Y 439.761,Z 280.015,A -85,B 0,C 180,E1 -9000,E2 -9000} C_VEL
LIN {X 0,Y 439.652,Z 280.023,A -85,B 0,C 180,E1 -9002.749,E2 -9002.749} C_VEL
LIN {X 0,Y 439.616,Z 280.033,A -85,B 0,C 180,E1 -9006.425,E2 -9006.425} C_VEL
LIN {X 0,Y 439.497,Z 280.041,A -85,B 0,C 180,E1 -9009.202,E2 -9009.202} C_VEL
LIN {X 0,Y 439.463,Z 280.056,A -85,B 0,C 180,E1 -9012.938,E2 -9012.938} C_VEL
LIN {X 0,Y 439.444,Z 280.056,A -85,B 0,C 180,E1 -9016.349,E2 -9016.349} C_VEL
LIN {X 0,Y 439.399,Z 280.063,A -85,B 0,C 180,E1 -9019.626,E2 -9019.626} C_VEL
LIN {X 0,Y 439.362,Z 280.069,A -85,B 0,C 180,E1 -9022.575,E2 -9022.575} C_VEL
LIN {X 0,Y 439.402,Z 280.064,A -85,B 0,C 180,E1 -9025.585,E2 -9025.585} C_VEL
LIN {X 0,Y 439.414,Z 280.066,A -85,B 0,C 180,E1 -9028.673,E2 -9028.673} C_VEL
LIN {X 0,Y 439.367,Z 280.069,A -85,B 0,C 180,E1 -9032.03,E2 -9032.03} C_VEL
LIN {X 0,Y 439.393,Z 280.064,A -85,B 0,C 180,E1 -9035.341,E2 -9035.341} C_VEL
LIN {X 0,Y 439.381,Z 280.073,A -85,B 0,C 180,E1 -9038.595,E2 -9038.595} C_VEL
LIN {X 0,Y 439.385,Z 280.069,A -85,B 0,C 180,E1 -9041.257,E2 -9041.257} C_VEL
LIN {X 0,Y 439.399,Z 280.069,A -85,B 0,C 180,E1 -9044.729,E2 -9044.729} C_VEL
LIN {X 0,Y 439.395,Z 280.065,A -85,B 0,C 180,E1 -9047.796,E2 -9047.796} C_VEL
LIN {X 0,Y 439.434,Z 280.061,A -85,B 0,C 180,E1 -9050.229,E2 -9050.229} C_VEL
LIN {X 0,Y 439.371,Z 280.069,A -85,B 0,C 180,E1 -9053.713,E2 -9053.713} C_VEL
LIN {X 0,Y 439.396,Z 280.112,A -85,B 0,C 180,E1 -9054.844,E2 -9054.844} C_VEL
LIN {X 0,Y 445.177,Z 298.059,A -85,B 0,C 180,E1 -9057.537,E2 -9057.537} C_VEL
LIN {X 0,Y 448.391,Z 308.778,A -85,B 0,C 180,E1 -9059.026,E2 -9059.026} C_VEL
LIN {X 0,Y 450.972,Z 314.547,A -85,B 0,C 180,E1 -9059.326,E2 -9059.326} C_VEL
LIN {X 0,Y 455.158,Z 338.707,A -85,B 0,C 180,E1 -9060.067,E2 -9060.067} C_VEL
LIN {X 0,Y 452.072,Z 515.782,A -85,B 0,C 180,E1 -9063.004,E2 -9063.004} C_VEL
LIN {X 0,Y 451.238,Z 531.978,A -85,B 0,C 180,E1 -9063.43,E2 -9063.43} C_VEL
LIN {X 0,Y 450.277,Z 547.839,A -85,B 0,C 180,E1 -9064.024,E2 -9064.024} C_VEL
LIN {X 0,Y 449.165,Z 563.04,A -85,B 0,C 180,E1 -9064.763,E2 -9064.763} C_VEL
LIN {X 0,Y 447.894,Z 578.449,A -85,B 0,C 180,E1 -9065.706,E2 -9065.706} C_VEL
LIN {X 0,Y 446.366,Z 593.307,A -85,B 0,C 180,E1 -9066.82,E2 -9066.82} C_VEL
LIN {X 0,Y 444.958,Z 607.317,A -85,B 0,C 180,E1 -9068.09,E2 -9068.09} C_VEL
LIN {X 0,Y 443.507,Z 621.252,A -85,B 0,C 180,E1 -9069.597,E2 -9069.597} C_VEL
LIN {X 0,Y 442.384,Z 632.269,A -85,B 0,C 180,E1 -9070.994,E2 -9070.994} C_VEL
LIN {X 0,Y 441.155,Z 644.332,A -85,B 0,C 180,E1 -9072.796,E2 -9072.796} C_VEL
LIN {X 0,Y 440.285,Z 653.87,A -85,B 0,C 180,E1 -9074.492,E2 -9074.492} C_VEL
LIN {X 0,Y 439.504,Z 662.79,A -85,B 0,C 180,E1 -9076.358,E2 -9076.358} C_VEL
LIN {X 0,Y 439.103,Z 669.44,A -85,B 0,C 180,E1 -9077.991,E2 -9077.991} C_VEL
LIN {X 0,Y 438.574,Z 677.132,A -85,B 0,C 180,E1 -9080.314,E2 -9080.314} C_VEL
LIN {X 0,Y 438.392,Z 682.989,A -85,B 0,C 180,E1 -9082.632,E2 -9082.632} C_VEL
LIN {X 0,Y 438.307,Z 686.415,A -85,B 0,C 180,E1 -9084.479,E2 -9084.479} C_VEL
LIN {X 0,Y 438.254,Z 688.904,A -85,B 0,C 180,E1 -9086.322,E2 -9086.322} C_VEL
LIN {X 0,Y 438.269,Z 690.31,A -85,B 0,C 180,E1 -9088.162,E2 -9088.162} C_VEL
LIN {X 0,Y 438.249,Z 690.839,A -85,B 0,C 180,E1 -9090,E2 -9090} C_VEL
LIN {X 0,Y 438.269,Z 690.309,A -85,B 0,C 180,E1 -9091.838,E2 -9091.838} C_VEL
LIN {X 0,Y 438.254,Z 688.901,A -85,B 0,C 180,E1 -9093.678,E2 -9093.678} C_VEL
LIN {X 0,Y 438.307,Z 686.412,A -85,B 0,C 180,E1 -9095.521,E2 -9095.521} C_VEL
LIN {X 0,Y 438.392,Z 682.989,A -85,B 0,C 180,E1 -9097.368,E2 -9097.368} C_VEL
LIN {X 0,Y 438.574,Z 677.13,A -85,B 0,C 180,E1 -9099.687,E2 -9099.687} C_VEL
LIN {X 0,Y 439.108,Z 669.434,A -85,B 0,C 180,E1 -9102.009,E2 -9102.009} C_VEL
LIN {X 0,Y 439.654,Z 660.745,A -85,B 0,C 180,E1 -9104.109,E2 -9104.109} C_VEL
LIN {X 0,Y 440.576,Z 651.378,A -85,B 0,C 180,E1 -9105.972,E2 -9105.972} C_VEL
LIN {X 0,Y 441.429,Z 641.738,A -85,B 0,C 180,E1 -9107.608,E2 -9107.608} C_VEL
LIN {X 0,Y 442.611,Z 630.514,A -85,B 0,C 180,E1 -9109.237,E2 -9109.237} C_VEL
LIN {X 0,Y 443.898,Z 618.049,A -85,B 0,C 180,E1 -9110.776,E2 -9110.776} C_VEL
LIN {X 0,Y 445.223,Z 604.927,A -85,B 0,C 180,E1 -9112.14,E2 -9112.14} C_VEL
LIN {X 0,Y 446.493,Z 591.831,A -85,B 0,C 180,E1 -9113.296,E2 -9113.296} C_VEL
LIN {X 0,Y 447.92,Z 577.495,A -85,B 0,C 180,E1 -9114.355,E2 -9114.355} C_VEL
LIN {X 0,Y 449.266,Z 561.97,A -85,B 0,C 180,E1 -9115.293,E2 -9115.293} C_VEL
LIN {X 0,Y 450.413,Z 546.453,A -85,B 0,C 180,E1 -9116.03,E2 -9116.03} C_VEL
LIN {X 0,Y 451.268,Z 530.94,A -85,B 0,C 180,E1 -9116.599,E2 -9116.599} C_VEL
LIN {X 0,Y 452.054,Z 514.324,A -85,B 0,C 180,E1 -9117.023,E2 -9117.023} C_VEL
LIN {X 0,Y 454.797,Z 357.647,A -85,B 0,C 180,E1 -9119.617,E2 -9119.617} C_VEL
LIN {X 0,Y 455.137,Z 338.757,A -85,B 0,C 180,E1 -9119.929,E2 -9119.929} C_VEL
LIN {X 0,Y 450.666,Z 313.678,A -85,B 0,C 180,E1 -9120.707,E2 -9120.707} C_VEL
LIN {X 0,Y 448.166,Z 308.142,A -85,B 0,C 180,E1 -9121.022,E2 -9121.022} C_VEL
LIN {X 0,Y 443.444,Z 292.418,A -85,B 0,C 180,E1 -9123.279,E2 -9123.279} C_VEL
LIN {X 0,Y 439.397,Z 280.065,A -85,B 0,C 180,E1 -9125.156,E2 -9125.156} C_VEL
LIN {X 0,Y 439.383,Z 280.067,A -85,B 0,C 180,E1 -9128.595,E2 -9128.595} C_VEL
LIN {X 0,Y 439.387,Z 280.066,A -85,B 0,C 180,E1 -9131.257,E2 -9131.257} C_VEL
LIN {X 0,Y 439.403,Z 280.06,A -85,B 0,C 180,E1 -9134.729,E2 -9134.729} C_VEL
LIN {X 0,Y 439.393,Z 280.059,A -85,B 0,C 180,E1 -9137.796,E2 -9137.796} C_VEL
LIN {X 0,Y 439.408,Z 280.056,A -85,B 0,C 180,E1 -9140.226,E2 -9140.226} C_VEL
LIN {X 0,Y 439.372,Z 280.064,A -85,B 0,C 180,E1 -9143.713,E2 -9143.713} C_VEL
LIN {X 0,Y 439.37,Z 280.066,A -85,B 0,C 180,E1 -9147.054,E2 -9147.054} C_VEL
LIN {X 0,Y 439.379,Z 280.061,A -85,B 0,C 180,E1 -9150.274,E2 -9150.274} C_VEL
LIN {X 0,Y 439.426,Z 280.063,A -85,B 0,C 180,E1 -9153.396,E2 -9153.396} C_VEL
LIN {X 0,Y 439.384,Z 280.063,A -85,B 0,C 180,E1 -9156.43,E2 -9156.43} C_VEL
LIN {X 0,Y 439.385,Z 280.049,A -85,B 0,C 180,E1 -9159.397,E2 -9159.397} C_VEL
LIN {X 0,Y 439.428,Z 280.056,A -85,B 0,C 180,E1 -9162.31,E2 -9162.31} C_VEL
LIN {X 0,Y 439.445,Z 280.047,A -85,B 0,C 180,E1 -9165.174,E2 -9165.174} C_VEL
LIN {X 0,Y 439.481,Z 280.045,A -85,B 0,C 180,E1 -9168.001,E2 -9168.001} C_VEL
LIN {X 0,Y 439.546,Z 280.036,A -85,B 0,C 180,E1 -9171.726,E2 -9171.726} C_VEL
LIN {X 0,Y 439.62,Z 280.019,A -85,B 0,C 180,E1 -9174.496,E2 -9174.496} C_VEL
LIN {X 0,Y 439.633,Z 280.031,A -85,B 0,C 180,E1 -9178.168,E2 -9178.168} C_VEL
LIN {X 0,Y 439.76,Z 280.002,A -85,B 0,C 180,E1 -9180,E2 -9180} C_VEL
LIN {X 0,Y 439.639,Z 280.025,A -85,B 0,C 180,E1 -9182.749,E2 -9182.749} C_VEL
LIN {X 0,Y 439.611,Z 280.032,A -85,B 0,C 180,E1 -9186.425,E2 -9186.425} C_VEL
LIN {X 0,Y 439.497,Z 280.037,A -85,B 0,C 180,E1 -9189.202,E2 -9189.202} C_VEL
LIN {X 0,Y 439.463,Z 280.054,A -85,B 0,C 180,E1 -9192.938,E2 -9192.938} C_VEL
LIN {X 0,Y 439.445,Z 280.043,A -85,B 0,C 180,E1 -9196.349,E2 -9196.349} C_VEL
LIN {X 0,Y 439.401,Z 280.059,A -85,B 0,C 180,E1 -9199.626,E2 -9199.626} C_VEL
LIN {X 0,Y 439.363,Z 280.051,A -85,B 0,C 180,E1 -9202.576,E2 -9202.576} C_VEL
LIN {X 0,Y 439.404,Z 280.06,A -85,B 0,C 180,E1 -9205.585,E2 -9205.585} C_VEL
LIN {X 0,Y 439.416,Z 280.048,A -85,B 0,C 180,E1 -9208.674,E2 -9208.674} C_VEL
LIN {X 0,Y 439.368,Z 280.062,A -85,B 0,C 180,E1 -9212.031,E2 -9212.031} C_VEL
LIN {X 0,Y 439.395,Z 280.063,A -85,B 0,C 180,E1 -9215.341,E2 -9215.341} C_VEL
LIN {X 0,Y 439.376,Z 280.054,A -85,B 0,C 180,E1 -9218.596,E2 -9218.596} C_VEL
LIN {X 0,Y 439.387,Z 280.058,A -85,B 0,C 180,E1 -9221.257,E2 -9221.257} C_VEL
LIN {X 0,Y 439.4,Z 280.063,A -85,B 0,C 180,E1 -9224.729,E2 -9224.729} C_VEL
LIN {X 0,Y 439.395,Z 280.063,A -85,B 0,C 180,E1 -9227.796,E2 -9227.796} C_VEL
LIN {X 0,Y 439.429,Z 280.06,A -85,B 0,C 180,E1 -9230.228,E2 -9230.228} C_VEL
LIN {X 0,Y 439.373,Z 280.052,A -85,B 0,C 180,E1 -9233.713,E2 -9233.713} C_VEL
LIN {X 0,Y 439.372,Z 280.051,A -85,B 0,C 180,E1 -9237.054,E2 -9237.054} C_VEL
LIN {X 0,Y 439.403,Z 280.119,A -85,B 0,C 180,E1 -9237.459,E2 -9237.459} C_VEL
LIN {X 0,Y 441.534,Z 286.817,A -85,B 0,C 180,E1 -9238.548,E2 -9238.548} C_VEL
LIN {X 0,Y 452.447,Z 308.75,A -85,B 0,C 180,E1 -9239.793,E2 -9239.793} C_VEL
LIN {X 0,Y 455.36,Z 315.001,A -85,B 0,C 180,E1 -9240.12,E2 -9240.12} C_VEL
LIN {X 0,Y 452.575,Z 481.272,A -85,B 0,C 180,E1 -9242.866,E2 -9242.866} C_VEL
LIN {X 0,Y 452.144,Z 495.519,A -85,B 0,C 180,E1 -9243.143,E2 -9243.143} C_VEL
LIN {X 0,Y 451.407,Z 499.42,A -85,B 0,C 180,E1 -9243.2,E2 -9243.2} C_VEL
LIN {X 0,Y 445.671,Z 511.684,A -85,B 0,C 180,E1 -9243.23,E2 -9243.23} C_VEL
LIN {X 0,Y 444.931,Z 515.501,A -85,B 0,C 180,E1 -9243.34,E2 -9243.34} C_VEL
LIN {X 0,Y 443.924,Z 530.924,A -85,B 0,C 180,E1 -9244.002,E2 -9244.002} C_VEL
LIN {X 0,Y 442.661,Z 546.922,A -85,B 0,C 180,E1 -9244.889,E2 -9244.889} C_VEL
LIN {X 0,Y 441.3,Z 561.71,A -85,B 0,C 180,E1 -9245.915,E2 -9245.915} C_VEL
LIN {X 0,Y 439.892,Z 575.619,A -85,B 0,C 180,E1 -9247.081,E2 -9247.081} C_VEL
LIN {X 0,Y 438.439,Z 588.785,A -85,B 0,C 180,E1 -9248.391,E2 -9248.391} C_VEL
LIN {X 0,Y 437.138,Z 600.65,A -85,B 0,C 180,E1 -9249.778,E2 -9249.778} C_VEL
LIN {X 0,Y 435.727,Z 612.558,A -85,B 0,C 180,E1 -9251.425,E2 -9251.425} C_VEL
LIN {X 0,Y 434.625,Z 622.693,A -85,B 0,C 180,E1 -9253.078,E2 -9253.078} C_VEL
LIN {X 0,Y 433.542,Z 632.535,A -85,B 0,C 180,E1 -9254.967,E2 -9254.967} C_VEL
LIN {X 0,Y 432.737,Z 640.804,A -85,B 0,C 180,E1 -9256.858,E2 -9256.858} C_VEL
LIN {X 0,Y 432.191,Z 647.611,A -85,B 0,C 180,E1 -9258.747,E2 -9258.747} C_VEL
LIN {X 0,Y 431.725,Z 653.204,A -85,B 0,C 180,E1 -9260.631,E2 -9260.631} C_VEL
LIN {X 0,Y 431.508,Z 657.702,A -85,B 0,C 180,E1 -9262.513,E2 -9262.513} C_VEL
LIN {X 0,Y 431.354,Z 661.071,A -85,B 0,C 180,E1 -9264.39,E2 -9264.39} C_VEL
LIN {X 0,Y 431.214,Z 663.521,A -85,B 0,C 180,E1 -9266.262,E2 -9266.262} C_VEL
LIN {X 0,Y 431.22,Z 664.913,A -85,B 0,C 180,E1 -9268.132,E2 -9268.132} C_VEL
LIN {X 0,Y 431.164,Z 665.452,A -85,B 0,C 180,E1 -9270,E2 -9270} C_VEL
LIN {X 0,Y 431.219,Z 664.96,A -85,B 0,C 180,E1 -9271.868,E2 -9271.868} C_VEL
LIN {X 0,Y 431.213,Z 663.615,A -85,B 0,C 180,E1 -9273.738,E2 -9273.738} C_VEL
LIN {X 0,Y 431.354,Z 661.212,A -85,B 0,C 180,E1 -9275.61,E2 -9275.61} C_VEL
LIN {X 0,Y 431.499,Z 657.901,A -85,B 0,C 180,E1 -9277.487,E2 -9277.487} C_VEL
LIN {X 0,Y 431.796,Z 652.213,A -85,B 0,C 180,E1 -9279.84,E2 -9279.84} C_VEL
LIN {X 0,Y 432.271,Z 646.328,A -85,B 0,C 180,E1 -9281.726,E2 -9281.726} C_VEL
LIN {X 0,Y 432.919,Z 639.232,A -85,B 0,C 180,E1 -9283.615,E2 -9283.615} C_VEL
LIN {X 0,Y 433.755,Z 630.738,A -85,B 0,C 180,E1 -9285.506,E2 -9285.506} C_VEL
LIN {X 0,Y 434.86,Z 620.58,A -85,B 0,C 180,E1 -9287.387,E2 -9287.387} C_VEL
LIN {X 0,Y 436.03,Z 609.95,A -85,B 0,C 180,E1 -9289.05,E2 -9289.05} C_VEL
LIN {X 0,Y 437.437,Z 597.526,A -85,B 0,C 180,E1 -9290.699,E2 -9290.699} C_VEL
LIN {X 0,Y 438.88,Z 584.993,A -85,B 0,C 180,E1 -9292.106,E2 -9292.106} C_VEL
LIN {X 0,Y 440.359,Z 571.45,A -85,B 0,C 180,E1 -9293.39,E2 -9293.39} C_VEL
LIN {X 0,Y 441.892,Z 556.376,A -85,B 0,C 180,E1 -9294.569,E2 -9294.569} C_VEL
LIN {X 0,Y 442.913,Z 544.177,A -85,B 0,C 180,E1 -9295.367,E2 -9295.367} C_VEL
LIN {X 0,Y 444.095,Z 529.21,A -85,B 0,C 180,E1 -9296.176,E2 -9296.176} C_VEL
LIN {X 0,Y 445.124,Z 511.695,A -85,B 0,C 180,E1 -9296.901,E2 -9296.901} C_VEL
LIN {X 0,Y 445.879,Z 495.721,A -85,B 0,C 180,E1 -9297.362,E2 -9297.362} C_VEL
LIN {X 0,Y 446.453,Z 471.601,A -85,B 0,C 180,E1 -9297.809,E2 -9297.809} C_VEL
LIN {X 0,Y 449.326,Z 317.382,A -85,B 0,C 180,E1 -9300.38,E2 -9300.38} C_VEL
LIN {X 0,Y 439.747,Z 297.453,A -85,B 0,C 180,E1 -9301.494,E2 -9301.494} C_VEL
LIN {X 0,Y 434.173,Z 286.838,A -85,B 0,C 180,E1 -9302.167,E2 -9302.167} C_VEL
LIN {X 0,Y 432.328,Z 280.935,A -85,B 0,C 180,E1 -9303.169,E2 -9303.169} C_VEL
LIN {X 0,Y 432.336,Z 280.93,A -85,B 0,C 180,E1 -9305.818,E2 -9305.818} C_VEL
LIN {X 0,Y 432.327,Z 280.943,A -85,B 0,C 180,E1 -9309.345,E2 -9309.345} C_VEL
LIN {X 0,Y 432.332,Z 280.941,A -85,B 0,C 180,E1 -9311.797,E2 -9311.797} C_VEL
LIN {X 0,Y 432.332,Z 280.943,A -85,B 0,C 180,E1 -9314.347,E2 -9314.347} C_VEL
LIN {X 0,Y 432.319,Z 280.946,A -85,B 0,C 180,E1 -9317.015,E2 -9317.015} C_VEL
LIN {X 0,Y 432.331,Z 280.942,A -85,B 0,C 180,E1 -9319.82,E2 -9319.82} C_VEL
LIN {X 0,Y 432.305,Z 280.94,A -85,B 0,C 180,E1 -9323.022,E2 -9323.022} C_VEL
LIN {X 0,Y 432.358,Z 280.937,A -85,B 0,C 180,E1 -9325.996,E2 -9325.996} C_VEL
LIN {X 0,Y 432.345,Z 280.944,A -85,B 0,C 180,E1 -9329.489,E2 -9329.489} C_VEL
LIN {X 0,Y 432.389,Z 280.925,A -85,B 0,C 180,E1 -9332.928,E2 -9332.928} C_VEL
LIN {X 0,Y 432.369,Z 280.935,A -85,B 0,C 180,E1 -9336.023,E2 -9336.023} C_VEL
LIN {X 0,Y 432.348,Z 280.932,A -85,B 0,C 180,E1 -9339.046,E2 -9339.046} C_VEL
LIN {X 0,Y 432.375,Z 280.934,A -85,B 0,C 180,E1 -9342.011,E2 -9342.011} C_VEL
LIN {X 0,Y 432.393,Z 280.922,A -85,B 0,C 180,E1 -9344.926,E2 -9344.926} C_VEL
LIN {X 0,Y 432.456,Z 280.925,A -85,B 0,C 180,E1 -9347.803,E2 -9347.803} C_VEL
LIN {X 0,Y 432.489,Z 280.916,A -85,B 0,C 180,E1 -9351.59,E2 -9351.59} C_VEL
LIN {X 0,Y 432.596,Z 280.91,A -85,B 0,C 180,E1 -9354.406,E2 -9354.406} C_VEL
LIN {X 0,Y 432.601,Z 280.896,A -85,B 0,C 180,E1 -9358.138,E2 -9358.138} C_VEL
LIN {X 0,Y 432.731,Z 280.891,A -85,B 0,C 180,E1 -9360,E2 -9360} C_VEL
LIN {X 0,Y 432.602,Z 280.899,A -85,B 0,C 180,E1 -9362.793,E2 -9362.793} C_VEL
LIN {X 0,Y 432.571,Z 280.911,A -85,B 0,C 180,E1 -9366.53,E2 -9366.53} C_VEL
LIN {X 0,Y 432.44,Z 280.918,A -85,B 0,C 180,E1 -9369.353,E2 -9369.353} C_VEL
LIN {X 0,Y 432.428,Z 280.93,A -85,B 0,C 180,E1 -9372.803,E2 -9372.803} C_VEL
LIN {X 0,Y 432.41,Z 280.933,A -85,B 0,C 180,E1 -9376.479,E2 -9376.479} C_VEL
LIN {X 0,Y 432.336,Z 280.942,A -85,B 0,C 180,E1 -9379.96,E2 -9379.96} C_VEL
LIN {X 0,Y 432.316,Z 280.951,A -85,B 0,C 180,E1 -9382.964,E2 -9382.964} C_VEL
LIN {X 0,Y 432.361,Z 280.941,A -85,B 0,C 180,E1 -9386.032,E2 -9386.032} C_VEL
LIN {X 0,Y 432.34,Z 280.945,A -85,B 0,C 180,E1 -9389.187,E2 -9389.187} C_VEL
LIN {X 0,Y 432.32,Z 280.95,A -85,B 0,C 180,E1 -9392.443,E2 -9392.443} C_VEL
LIN {X 0,Y 432.343,Z 280.942,A -85,B 0,C 180,E1 -9395.632,E2 -9395.632} C_VEL
LIN {X 0,Y 432.344,Z 280.949,A -85,B 0,C 180,E1 -9398.716,E2 -9398.716} C_VEL
LIN {X 0,Y 432.33,Z 280.946,A -85,B 0,C 180,E1 -9401.797,E2 -9401.797} C_VEL
LIN {X 0,Y 432.331,Z 280.948,A -85,B 0,C 180,E1 -9404.347,E2 -9404.347} C_VEL
LIN {X 0,Y 432.322,Z 280.95,A -85,B 0,C 180,E1 -9407.015,E2 -9407.015} C_VEL
LIN {X 0,Y 432.339,Z 280.944,A -85,B 0,C 180,E1 -9409.82,E2 -9409.82} C_VEL
LIN {X 0,Y 432.304,Z 280.946,A -85,B 0,C 180,E1 -9413.022,E2 -9413.022} C_VEL
LIN {X 0,Y 432.356,Z 281.07,A -85,B 0,C 180,E1 -9414.337,E2 -9414.337} C_VEL
LIN {X 0,Y 437.851,Z 297.82,A -85,B 0,C 180,E1 -9416.925,E2 -9416.925} C_VEL
LIN {X 0,Y 440.996,Z 308.188,A -85,B 0,C 180,E1 -9418.441,E2 -9418.441} C_VEL
LIN {X 0,Y 445.162,Z 317.43,A -85,B 0,C 180,E1 -9418.938,E2 -9418.938} C_VEL
LIN {X 0,Y 448.985,Z 340.065,A -85,B 0,C 180,E1 -9419.64,E2 -9419.64} C_VEL
LIN {X 0,Y 445.735,Z 515.872,A -85,B 0,C 180,E1 -9422.594,E2 -9422.594} C_VEL
LIN {X 0,Y 444.843,Z 531.778,A -85,B 0,C 180,E1 -9423.017,E2 -9423.017} C_VEL
LIN {X 0,Y 443.898,Z 547.638,A -85,B 0,C 180,E1 -9423.622,E2 -9423.622} C_VEL
LIN {X 0,Y 442.719,Z 562.837,A -85,B 0,C 180,E1 -9424.369,E2 -9424.369} C_VEL
LIN {X 0,Y 441.402,Z 578.151,A -85,B 0,C 180,E1 -9425.318,E2 -9425.318} C_VEL
LIN {X 0,Y 439.804,Z 593.102,A -85,B 0,C 180,E1 -9426.454,E2 -9426.454} C_VEL
LIN {X 0,Y 438.317,Z 607.111,A -85,B 0,C 180,E1 -9427.741,E2 -9427.741} C_VEL
LIN {X 0,Y 436.926,Z 619.847,A -85,B 0,C 180,E1 -9429.125,E2 -9429.125} C_VEL
LIN {X 0,Y 435.583,Z 632.06,A -85,B 0,C 180,E1 -9430.685,E2 -9430.685} C_VEL
LIN {X 0,Y 434.379,Z 643.03,A -85,B 0,C 180,E1 -9432.339,E2 -9432.339} C_VEL
LIN {X 0,Y 433.526,Z 652.421,A -85,B 0,C 180,E1 -9434.003,E2 -9434.003} C_VEL
LIN {X 0,Y 432.595,Z 661.563,A -85,B 0,C 180,E1 -9435.896,E2 -9435.896} C_VEL
LIN {X 0,Y 432.079,Z 669.231,A -85,B 0,C 180,E1 -9437.793,E2 -9437.793} C_VEL
LIN {X 0,Y 431.496,Z 676.923,A -85,B 0,C 180,E1 -9440.153,E2 -9440.153} C_VEL
LIN {X 0,Y 431.312,Z 682.781,A -85,B 0,C 180,E1 -9442.51,E2 -9442.51} C_VEL
LIN {X 0,Y 431.22,Z 686.207,A -85,B 0,C 180,E1 -9444.388,E2 -9444.388} C_VEL
LIN {X 0,Y 431.16,Z 688.697,A -85,B 0,C 180,E1 -9446.262,E2 -9446.262} C_VEL
LIN {X 0,Y 431.193,Z 690.104,A -85,B 0,C 180,E1 -9448.132,E2 -9448.132} C_VEL
LIN {X 0,Y 431.163,Z 690.632,A -85,B 0,C 180,E1 -9450,E2 -9450} C_VEL
LIN {X 0,Y 431.193,Z 690.102,A -85,B 0,C 180,E1 -9451.868,E2 -9451.868} C_VEL
LIN {X 0,Y 431.16,Z 688.694,A -85,B 0,C 180,E1 -9453.738,E2 -9453.738} C_VEL
LIN {X 0,Y 431.22,Z 686.204,A -85,B 0,C 180,E1 -9455.612,E2 -9455.612} C_VEL
LIN {X 0,Y 431.312,Z 682.78,A -85,B 0,C 180,E1 -9457.49,E2 -9457.49} C_VEL
LIN {X 0,Y 431.496,Z 676.92,A -85,B 0,C 180,E1 -9459.847,E2 -9459.847} C_VEL
LIN {X 0,Y 432.085,Z 669.223,A -85,B 0,C 180,E1 -9462.207,E2 -9462.207} C_VEL
LIN {X 0,Y 432.666,Z 660.534,A -85,B 0,C 180,E1 -9464.342,E2 -9464.342} C_VEL
LIN {X 0,Y 433.61,Z 651.164,A -85,B 0,C 180,E1 -9466.236,E2 -9466.236} C_VEL
LIN {X 0,Y 434.546,Z 641.525,A -85,B 0,C 180,E1 -9467.896,E2 -9467.896} C_VEL
LIN {X 0,Y 435.801,Z 630.301,A -85,B 0,C 180,E1 -9469.55,E2 -9469.55} C_VEL
LIN {X 0,Y 437.082,Z 618.622,A -85,B 0,C 180,E1 -9471.017,E2 -9471.017} C_VEL
LIN {X 0,Y 438.431,Z 605.893,A -85,B 0,C 180,E1 -9472.378,E2 -9472.378} C_VEL
LIN {X 0,Y 439.935,Z 591.618,A -85,B 0,C 180,E1 -9473.664,E2 -9473.664} C_VEL
LIN {X 0,Y 441.388,Z 577.281,A -85,B 0,C 180,E1 -9474.739,E2 -9474.739} C_VEL
LIN {X 0,Y 442.808,Z 561.756,A -85,B 0,C 180,E1 -9475.689,E2 -9475.689} C_VEL
LIN {X 0,Y 444.008,Z 546.238,A -85,B 0,C 180,E1 -9476.435,E2 -9476.435} C_VEL
LIN {X 0,Y 444.931,Z 530.723,A -85,B 0,C 180,E1 -9477.009,E2 -9477.009} C_VEL
LIN {X 0,Y 445.726,Z 514.547,A -85,B 0,C 180,E1 -9477.43,E2 -9477.43} C_VEL
LIN {X 0,Y 448.621,Z 358.681,A -85,B 0,C 180,E1 -9480.044,E2 -9480.044} C_VEL
LIN {X 0,Y 448.835,Z 339.095,A -85,B 0,C 180,E1 -9480.382,E2 -9480.382} C_VEL
LIN {X 0,Y 444.846,Z 316.507,A -85,B 0,C 180,E1 -9481.097,E2 -9481.097} C_VEL
LIN {X 0,Y 440.972,Z 308.114,A -85,B 0,C 180,E1 -9481.559,E2 -9481.559} C_VEL
LIN {X 0,Y 435.479,Z 290.328,A -85,B 0,C 180,E1 -9484.199,E2 -9484.199} C_VEL
LIN {X 0,Y 432.346,Z 280.946,A -85,B 0,C 180,E1 -9485.683,E2 -9485.683} C_VEL
LIN {X 0,Y 432.353,Z 280.942,A -85,B 0,C 180,E1 -9489.342,E2 -9489.342} C_VEL
LIN {X 0,Y 432.333,Z 280.944,A -85,B 0,C 180,E1 -9491.797,E2 -9491.797} C_VEL
LIN {X 0,Y 432.338,Z 280.939,A -85,B 0,C 180,E1 -9494.346,E2 -9494.346} C_VEL
LIN {X 0,Y 432.318,Z 280.944,A -85,B 0,C 180,E1 -9497.016,E2 -9497.016} C_VEL
LIN {X 0,Y 432.33,Z 280.938,A -85,B 0,C 180,E1 -9499.821,E2 -9499.821} C_VEL
LIN {X 0,Y 432.304,Z 280.944,A -85,B 0,C 180,E1 -9503.022,E2 -9503.022} C_VEL
LIN {X 0,Y 432.357,Z 280.937,A -85,B 0,C 180,E1 -9505.996,E2 -9505.996} C_VEL
LIN {X 0,Y 432.345,Z 280.94,A -85,B 0,C 180,E1 -9509.49,E2 -9509.49} C_VEL
LIN {X 0,Y 432.388,Z 280.936,A -85,B 0,C 180,E1 -9512.928,E2 -9512.928} C_VEL
LIN {X 0,Y 432.369,Z 280.936,A -85,B 0,C 180,E1 -9516.023,E2 -9516.023} C_VEL
LIN {X 0,Y 432.347,Z 280.93,A -85,B 0,C 180,E1 -9519.046,E2 -9519.046} C_VEL
LIN {X 0,Y 432.375,Z 280.934,A -85,B 0,C 180,E1 -9522.011,E2 -9522.011} C_VEL
LIN {X 0,Y 432.393,Z 280.929,A -85,B 0,C 180,E1 -9524.927,E2 -9524.927} C_VEL
LIN {X 0,Y 432.457,Z 280.92,A -85,B 0,C 180,E1 -9527.804,E2 -9527.804} C_VEL
LIN {X 0,Y 432.49,Z 280.916,A -85,B 0,C 180,E1 -9531.59,E2 -9531.59} C_VEL
LIN {X 0,Y 432.596,Z 280.893,A -85,B 0,C 180,E1 -9534.406,E2 -9534.406} C_VEL
LIN {X 0,Y 432.603,Z 280.906,A -85,B 0,C 180,E1 -9538.138,E2 -9538.138} C_VEL
LIN {X 0,Y 432.73,Z 280.877,A -85,B 0,C 180,E1 -9540,E2 -9540} C_VEL
LIN {X 0,Y 432.591,Z 280.903,A -85,B 0,C 180,E1 -9542.794,E2 -9542.794} C_VEL
LIN {X 0,Y 432.567,Z 280.908,A -85,B 0,C 180,E1 -9546.531,E2 -9546.531} C_VEL
LIN {X 0,Y 432.44,Z 280.918,A -85,B 0,C 180,E1 -9549.353,E2 -9549.353} C_VEL
LIN {X 0,Y 432.429,Z 280.932,A -85,B 0,C 180,E1 -9552.804,E2 -9552.804} C_VEL
LIN {X 0,Y 432.411,Z 280.92,A -85,B 0,C 180,E1 -9556.479,E2 -9556.479} C_VEL
LIN {X 0,Y 432.337,Z 280.938,A -85,B 0,C 180,E1 -9559.961,E2 -9559.961} C_VEL
LIN {X 0,Y 432.318,Z 280.933,A -85,B 0,C 180,E1 -9562.964,E2 -9562.964} C_VEL
LIN {X 0,Y 432.362,Z 280.936,A -85,B 0,C 180,E1 -9566.033,E2 -9566.033} C_VEL
LIN {X 0,Y 432.341,Z 280.937,A -85,B 0,C 180,E1 -9569.188,E2 -9569.188} C_VEL
LIN {X 0,Y 432.321,Z 280.942,A -85,B 0,C 180,E1 -9572.443,E2 -9572.443} C_VEL
LIN {X 0,Y 432.344,Z 280.94,A -85,B 0,C 180,E1 -9575.632,E2 -9575.632} C_VEL
LIN {X 0,Y 432.339,Z 280.931,A -85,B 0,C 180,E1 -9578.715,E2 -9578.715} C_VEL
LIN {X 0,Y 432.332,Z 280.933,A -85,B 0,C 180,E1 -9581.797,E2 -9581.797} C_VEL
LIN {X 0,Y 432.333,Z 280.944,A -85,B 0,C 180,E1 -9584.348,E2 -9584.348} C_VEL
LIN {X 0,Y 432.32,Z 280.945,A -85,B 0,C 180,E1 -9587.016,E2 -9587.016} C_VEL
LIN {X 0,Y 432.336,Z 280.942,A -85,B 0,C 180,E1 -9589.821,E2 -9589.821} C_VEL
LIN {X 0,Y 432.306,Z 280.926,A -85,B 0,C 180,E1 -9593.022,E2 -9593.022} C_VEL
LIN {X 0,Y 432.359,Z 280.93,A -85,B 0,C 180,E1 -9595.997,E2 -9595.997} C_VEL
LIN {X 0,Y 432.35,Z 281.012,A -85,B 0,C 180,E1 -9596.955,E2 -9596.955} C_VEL
LIN {X 0,Y 434.244,Z 287.102,A -85,B 0,C 180,E1 -9597.957,E2 -9597.957} C_VEL
LIN {X 0,Y 443.711,Z 305.47,A -85,B 0,C 180,E1 -9599.067,E2 -9599.067} C_VEL
LIN {X 0,Y 449.285,Z 317.563,A -85,B 0,C 180,E1 -9599.716,E2 -9599.716} C_VEL
LIN {X 0,Y 446.086,Z 489.031,A -85,B 0,C 180,E1 -9602.589,E2 -9602.589} C_VEL
LIN {X 0,Y 445.443,Z 505.347,A -85,B 0,C 180,E1 -9602.993,E2 -9602.993} C_VEL
LIN {X 0,Y 444.931,Z 515.501,A -85,B 0,C 180,E1 -9603.34,E2 -9603.34} C_VEL
LIN {X 0,Y 444.116,Z 521.331,A -85,B 0,C 180,E1 -9603.535,E2 -9603.535} C_VEL
LIN {X 0,Y 438.109,Z 537.772,A -85,B 0,C 180,E1 -9604.011,E2 -9604.011} C_VEL
LIN {X 0,Y 436.678,Z 543.036,A -85,B 0,C 180,E1 -9604.253,E2 -9604.253} C_VEL
LIN {X 0,Y 436.448,Z 544.786,A -85,B 0,C 180,E1 -9604.352,E2 -9604.352} C_VEL
LIN {X 0,Y 435.147,Z 558.772,A -85,B 0,C 180,E1 -9605.298,E2 -9605.298} C_VEL
LIN {X 0,Y 433.776,Z 571.977,A -85,B 0,C 180,E1 -9606.36,E2 -9606.36} C_VEL
LIN {X 0,Y 432.222,Z 585.482,A -85,B 0,C 180,E1 -9607.661,E2 -9607.661} C_VEL
LIN {X 0,Y 430.824,Z 596.995,A -85,B 0,C 180,E1 -9608.968,E2 -9608.968} C_VEL
LIN {X 0,Y 429.505,Z 607.926,A -85,B 0,C 180,E1 -9610.401,E2 -9610.401} C_VEL
LIN {X 0,Y 428.147,Z 619.444,A -85,B 0,C 180,E1 -9612.188,E2 -9612.188} C_VEL
LIN {X 0,Y 427.005,Z 629.261,A -85,B 0,C 180,E1 -9613.997,E2 -9613.997} C_VEL
LIN {X 0,Y 426.161,Z 637.061,A -85,B 0,C 180,E1 -9615.678,E2 -9615.678} C_VEL
LIN {X 0,Y 425.414,Z 644.594,A -85,B 0,C 180,E1 -9617.598,E2 -9617.598} C_VEL
LIN {X 0,Y 424.839,Z 650.758,A -85,B 0,C 180,E1 -9619.516,E2 -9619.516} C_VEL
LIN {X 0,Y 424.565,Z 655.806,A -85,B 0,C 180,E1 -9621.432,E2 -9621.432} C_VEL
LIN {X 0,Y 424.345,Z 660.141,A -85,B 0,C 180,E1 -9623.575,E2 -9623.575} C_VEL
LIN {X 0,Y 424.186,Z 662.622,A -85,B 0,C 180,E1 -9625.248,E2 -9625.248} C_VEL
LIN {X 0,Y 424.192,Z 664.529,A -85,B 0,C 180,E1 -9627.151,E2 -9627.151} C_VEL
LIN {X 0,Y 424.088,Z 665.502,A -85,B 0,C 180,E1 -9629.05,E2 -9629.05} C_VEL
LIN {X 0,Y 424.088,Z 665.518,A -85,B 0,C 180,E1 -9630.95,E2 -9630.95} C_VEL
LIN {X 0,Y 424.192,Z 664.607,A -85,B 0,C 180,E1 -9632.849,E2 -9632.849} C_VEL
LIN {X 0,Y 424.184,Z 662.731,A -85,B 0,C 180,E1 -9634.752,E2 -9634.752} C_VEL
LIN {X 0,Y 424.35,Z 659.883,A -85,B 0,C 180,E1 -9636.657,E2 -9636.657} C_VEL
LIN {X 0,Y 424.559,Z 656.007,A -85,B 0,C 180,E1 -9638.568,E2 -9638.568} C_VEL
LIN {X 0,Y 424.821,Z 651.028,A -85,B 0,C 180,E1 -9640.485,E2 -9640.485} C_VEL
LIN {X 0,Y 425.387,Z 644.934,A -85,B 0,C 180,E1 -9642.402,E2 -9642.402} C_VEL
LIN {X 0,Y 426.239,Z 636.447,A -85,B 0,C 180,E1 -9644.563,E2 -9644.563} C_VEL
LIN {X 0,Y 427.286,Z 627.285,A -85,B 0,C 180,E1 -9646.483,E2 -9646.483} C_VEL
LIN {X 0,Y 428.356,Z 617.857,A -85,B 0,C 180,E1 -9648.163,E2 -9648.163} C_VEL
LIN {X 0,Y 429.665,Z 606.859,A -85,B 0,C 180,E1 -9649.84,E2 -9649.84} C_VEL
LIN {X 0,Y 431.227,Z 593.882,A -85,B 0,C 180,E1 -9651.506,E2 -9651.506} C_VEL
LIN {X 0,Y 432.847,Z 580.528,A -85,B 0,C 180,E1 -9652.934,E2 -9652.934} C_VEL
LIN {X 0,Y 434.246,Z 567.414,A -85,B 0,C 180,E1 -9654.12,E2 -9654.12} C_VEL
LIN {X 0,Y 435.65,Z 553.559,A -85,B 0,C 180,E1 -9655.174,E2 -9655.174} C_VEL
LIN {X 0,Y 436.975,Z 538.428,A -85,B 0,C 180,E1 -9656.121,E2 -9656.121} C_VEL
LIN {X 0,Y 438.217,Z 522.928,A -85,B 0,C 180,E1 -9656.876,E2 -9656.876} C_VEL
LIN {X 0,Y 439.021,Z 507.368,A -85,B 0,C 180,E1 -9657.467,E2 -9657.467} C_VEL
LIN {X 0,Y 439.785,Z 490.723,A -85,B 0,C 180,E1 -9657.902,E2 -9657.902} C_VEL
LIN {X 0,Y 443.14,Z 319.478,A -85,B 0,C 180,E1 -9660.815,E2 -9660.815} C_VEL
LIN {X 0,Y 434.606,Z 301.626,A -85,B 0,C 180,E1 -9661.833,E2 -9661.833} C_VEL
LIN {X 0,Y 426.909,Z 287.079,A -85,B 0,C 180,E1 -9662.781,E2 -9662.781} C_VEL
LIN {X 0,Y 425.301,Z 281.815,A -85,B 0,C 180,E1 -9663.719,E2 -9663.719} C_VEL
LIN {X 0,Y 425.262,Z 281.806,A -85,B 0,C 180,E1 -9666.508,E2 -9666.508} C_VEL
LIN {X 0,Y 425.281,Z 281.823,A -85,B 0,C 180,E1 -9669.04,E2 -9669.04} C_VEL
LIN {X 0,Y 425.289,Z 281.817,A -85,B 0,C 180,E1 -9671.958,E2 -9671.958} C_VEL
LIN {X 0,Y 425.283,Z 281.817,A -85,B 0,C 180,E1 -9675.283,E2 -9675.283} C_VEL
LIN {X 0,Y 425.272,Z 281.818,A -85,B 0,C 180,E1 -9678.621,E2 -9678.621} C_VEL
LIN {X 0,Y 425.3,Z 281.823,A -85,B 0,C 180,E1 -9681.101,E2 -9681.101} C_VEL
LIN {X 0,Y 425.298,Z 281.818,A -85,B 0,C 180,E1 -9684.664,E2 -9684.664} C_VEL
LIN {X 0,Y 425.263,Z 281.817,A -85,B 0,C 180,E1 -9688.073,E2 -9688.073} C_VEL
LIN {X 0,Y 425.329,Z 281.807,A -85,B 0,C 180,E1 -9691.368,E2 -9691.368} C_VEL
LIN {X 0,Y 425.293,Z 281.818,A -85,B 0,C 180,E1 -9694.554,E2 -9694.554} C_VEL
LIN {X 0,Y 425.285,Z 281.805,A -85,B 0,C 180,E1 -9697.661,E2 -9697.661} C_VEL
LIN {X 0,Y 425.359,Z 281.812,A -85,B 0,C 180,E1 -9700.704,E2 -9700.704} C_VEL
LIN {X 0,Y 425.386,Z 281.789,A -85,B 0,C 180,E1 -9703.688,E2 -9703.688} C_VEL
LIN {X 0,Y 425.409,Z 281.804,A -85,B 0,C 180,E1 -9707.598,E2 -9707.598} C_VEL
LIN {X 0,Y 425.439,Z 281.791,A -85,B 0,C 180,E1 -9711.45,E2 -9711.45} C_VEL
LIN {X 0,Y 425.553,Z 281.787,A -85,B 0,C 180,E1 -9714.313,E2 -9714.313} C_VEL
LIN {X 0,Y 425.57,Z 281.771,A -85,B 0,C 180,E1 -9718.107,E2 -9718.107} C_VEL
LIN {X 0,Y 425.701,Z 281.767,A -85,B 0,C 180,E1 -9720,E2 -9720} C_VEL
LIN {X 0,Y 425.553,Z 281.776,A -85,B 0,C 180,E1 -9722.84,E2 -9722.84} C_VEL
LIN {X 0,Y 425.529,Z 281.789,A -85,B 0,C 180,E1 -9726.639,E2 -9726.639} C_VEL
LIN {X 0,Y 425.398,Z 281.794,A -85,B 0,C 180,E1 -9729.509,E2 -9729.509} C_VEL
LIN {X 0,Y 425.39,Z 281.808,A -85,B 0,C 180,E1 -9732.904,E2 -9732.904} C_VEL
LIN {X 0,Y 425.358,Z 281.813,A -85,B 0,C 180,E1 -9736.605,E2 -9736.605} C_VEL
LIN {X 0,Y 425.325,Z 281.816,A -85,B 0,C 180,E1 -9739.636,E2 -9739.636} C_VEL
LIN {X 0,Y 425.304,Z 281.82,A -85,B 0,C 180,E1 -9743.365,E2 -9743.365} C_VEL
LIN {X 0,Y 425.344,Z 281.817,A -85,B 0,C 180,E1 -9746.844,E2 -9746.844} C_VEL
LIN {X 0,Y 425.288,Z 281.821,A -85,B 0,C 180,E1 -9749.72,E2 -9749.72} C_VEL
LIN {X 0,Y 425.279,Z 281.825,A -85,B 0,C 180,E1 -9753.048,E2 -9753.048} C_VEL
LIN {X 0,Y 425.282,Z 281.821,A -85,B 0,C 180,E1 -9755.929,E2 -9755.929} C_VEL
LIN {X 0,Y 425.293,Z 281.827,A -85,B 0,C 180,E1 -9759.043,E2 -9759.043} C_VEL
LIN {X 0,Y 425.272,Z 281.829,A -85,B 0,C 180,E1 -9762.653,E2 -9762.653} C_VEL
LIN {X 0,Y 425.265,Z 281.826,A -85,B 0,C 180,E1 -9766.045,E2 -9766.045} C_VEL
LIN {X 0,Y 425.282,Z 281.824,A -85,B 0,C 180,E1 -9769.479,E2 -9769.479} C_VEL
LIN {X 0,Y 425.276,Z 281.825,A -85,B 0,C 180,E1 -9772.489,E2 -9772.489} C_VEL
LIN {X 0,Y 425.288,Z 281.924,A -85,B 0,C 180,E1 -9773.792,E2 -9773.792} C_VEL
LIN {X 0,Y 430.615,Z 297.944,A -85,B 0,C 180,E1 -9776.342,E2 -9776.342} C_VEL
LIN {X 0,Y 433.722,Z 307.926,A -85,B 0,C 180,E1 -9777.848,E2 -9777.848} C_VEL
LIN {X 0,Y 439.326,Z 320.205,A -85,B 0,C 180,E1 -9778.534,E2 -9778.534} C_VEL
LIN {X 0,Y 442.847,Z 341.286,A -85,B 0,C 180,E1 -9779.2,E2 -9779.2} C_VEL
LIN {X 0,Y 439.445,Z 515.948,A -85,B 0,C 180,E1 -9782.174,E2 -9782.174} C_VEL
LIN {X 0,Y 438.477,Z 532.497,A -85,B 0,C 180,E1 -9782.625,E2 -9782.625} C_VEL
LIN {X 0,Y 437.423,Z 548.74,A -85,B 0,C 180,E1 -9783.265,E2 -9783.265} C_VEL
LIN {X 0,Y 436.108,Z 564.625,A -85,B 0,C 180,E1 -9784.08,E2 -9784.08} C_VEL
LIN {X 0,Y 434.819,Z 578.878,A -85,B 0,C 180,E1 -9784.99,E2 -9784.99} C_VEL
LIN {X 0,Y 433.088,Z 594.328,A -85,B 0,C 180,E1 -9786.193,E2 -9786.193} C_VEL
LIN {X 0,Y 431.52,Z 608.083,A -85,B 0,C 180,E1 -9787.497,E2 -9787.497} C_VEL
LIN {X 0,Y 430.065,Z 620.837,A -85,B 0,C 180,E1 -9788.93,E2 -9788.93} C_VEL
LIN {X 0,Y 428.784,Z 631.852,A -85,B 0,C 180,E1 -9790.366,E2 -9790.366} C_VEL
LIN {X 0,Y 427.5,Z 642.98,A -85,B 0,C 180,E1 -9792.071,E2 -9792.071} C_VEL
LIN {X 0,Y 426.573,Z 652.211,A -85,B 0,C 180,E1 -9793.735,E2 -9793.735} C_VEL
LIN {X 0,Y 425.6,Z 661.354,A -85,B 0,C 180,E1 -9795.659,E2 -9795.659} C_VEL
LIN {X 0,Y 425.042,Z 669.022,A -85,B 0,C 180,E1 -9797.587,E2 -9797.587} C_VEL
LIN {X 0,Y 424.439,Z 676.714,A -85,B 0,C 180,E1 -9799.988,E2 -9799.988} C_VEL
LIN {X 0,Y 424.23,Z 682.573,A -85,B 0,C 180,E1 -9802.384,E2 -9802.384} C_VEL
LIN {X 0,Y 424.14,Z 686,A -85,B 0,C 180,E1 -9804.294,E2 -9804.294} C_VEL
LIN {X 0,Y 424.07,Z 688.49,A -85,B 0,C 180,E1 -9806.199,E2 -9806.199} C_VEL
LIN {X 0,Y 424.119,Z 689.897,A -85,B 0,C 180,E1 -9808.101,E2 -9808.101} C_VEL
LIN {X 0,Y 424.08,Z 690.425,A -85,B 0,C 180,E1 -9810,E2 -9810} C_VEL
LIN {X 0,Y 424.119,Z 689.895,A -85,B 0,C 180,E1 -9811.899,E2 -9811.899} C_VEL
LIN {X 0,Y 424.07,Z 688.486,A -85,B 0,C 180,E1 -9813.801,E2 -9813.801} C_VEL
LIN {X 0,Y 424.223,Z 685.109,A -85,B 0,C 180,E1 -9816.28,E2 -9816.28} C_VEL
LIN {X 0,Y 424.318,Z 680.414,A -85,B 0,C 180,E1 -9818.573,E2 -9818.573} C_VEL
LIN {X 0,Y 424.543,Z 675.276,A -85,B 0,C 180,E1 -9820.492,E2 -9820.492} C_VEL
LIN {X 0,Y 425.037,Z 669.012,A -85,B 0,C 180,E1 -9822.413,E2 -9822.413} C_VEL
LIN {X 0,Y 425.716,Z 660.323,A -85,B 0,C 180,E1 -9824.581,E2 -9824.581} C_VEL
LIN {X 0,Y 426.678,Z 650.952,A -85,B 0,C 180,E1 -9826.507,E2 -9826.507} C_VEL
LIN {X 0,Y 427.646,Z 641.311,A -85,B 0,C 180,E1 -9828.195,E2 -9828.195} C_VEL
LIN {X 0,Y 429.012,Z 630.088,A -85,B 0,C 180,E1 -9829.872,E2 -9829.872} C_VEL
LIN {X 0,Y 430.417,Z 617.657,A -85,B 0,C 180,E1 -9831.454,E2 -9831.454} C_VEL
LIN {X 0,Y 431.93,Z 604.501,A -85,B 0,C 180,E1 -9832.859,E2 -9832.859} C_VEL
LIN {X 0,Y 433.523,Z 589.972,A -85,B 0,C 180,E1 -9834.163,E2 -9834.163} C_VEL
LIN {X 0,Y 435.11,Z 575.001,A -85,B 0,C 180,E1 -9835.27,E2 -9835.27} C_VEL
LIN {X 0,Y 436.568,Z 559.318,A -85,B 0,C 180,E1 -9836.212,E2 -9836.212} C_VEL
LIN {X 0,Y 437.865,Z 543.385,A -85,B 0,C 180,E1 -9836.964,E2 -9836.964} C_VEL
LIN {X 0,Y 438.744,Z 528.672,A -85,B 0,C 180,E1 -9837.486,E2 -9837.486} C_VEL
LIN {X 0,Y 439.536,Z 511.506,A -85,B 0,C 180,E1 -9837.91,E2 -9837.91} C_VEL
LIN {X 0,Y 442.465,Z 358.634,A -85,B 0,C 180,E1 -9840.503,E2 -9840.503} C_VEL
LIN {X 0,Y 442.832,Z 341.157,A -85,B 0,C 180,E1 -9840.797,E2 -9840.797} C_VEL
LIN {X 0,Y 439.087,Z 319.399,A -85,B 0,C 180,E1 -9841.493,E2 -9841.493} C_VEL
LIN {X 0,Y 433.63,Z 307.746,A -85,B 0,C 180,E1 -9842.172,E2 -9842.172} C_VEL
LIN {X 0,Y 428.513,Z 291.461,A -85,B 0,C 180,E1 -9844.658,E2 -9844.658} C_VEL
LIN {X 0,Y 425.259,Z 281.826,A -85,B 0,C 180,E1 -9846.236,E2 -9846.236} C_VEL
LIN {X 0,Y 425.298,Z 281.822,A -85,B 0,C 180,E1 -9849.044,E2 -9849.044} C_VEL
LIN {X 0,Y 425.276,Z 281.821,A -85,B 0,C 180,E1 -9852.653,E2 -9852.653} C_VEL
LIN {X 0,Y 425.259,Z 281.819,A -85,B 0,C 180,E1 -9856.044,E2 -9856.044} C_VEL
LIN {X 0,Y 425.271,Z 281.817,A -85,B 0,C 180,E1 -9858.621,E2 -9858.621} C_VEL
LIN {X 0,Y 425.299,Z 281.817,A -85,B 0,C 180,E1 -9861.102,E2 -9861.102} C_VEL
LIN {X 0,Y 425.297,Z 281.817,A -85,B 0,C 180,E1 -9864.664,E2 -9864.664} C_VEL
LIN {X 0,Y 425.262,Z 281.821,A -85,B 0,C 180,E1 -9868.073,E2 -9868.073} C_VEL
LIN {X 0,Y 425.328,Z 281.818,A -85,B 0,C 180,E1 -9871.368,E2 -9871.368} C_VEL
LIN {X 0,Y 425.293,Z 281.82,A -85,B 0,C 180,E1 -9874.555,E2 -9874.555} C_VEL
LIN {X 0,Y 425.285,Z 281.819,A -85,B 0,C 180,E1 -9877.661,E2 -9877.661} C_VEL
LIN {X 0,Y 425.359,Z 281.794,A -85,B 0,C 180,E1 -9880.704,E2 -9880.704} C_VEL
LIN {X 0,Y 425.386,Z 281.807,A -85,B 0,C 180,E1 -9883.688,E2 -9883.688} C_VEL
LIN {X 0,Y 425.409,Z 281.795,A -85,B 0,C 180,E1 -9887.598,E2 -9887.598} C_VEL
LIN {X 0,Y 425.44,Z 281.795,A -85,B 0,C 180,E1 -9891.45,E2 -9891.45} C_VEL
LIN {X 0,Y 425.553,Z 281.769,A -85,B 0,C 180,E1 -9894.313,E2 -9894.313} C_VEL
LIN {X 0,Y 425.573,Z 281.782,A -85,B 0,C 180,E1 -9898.107,E2 -9898.107} C_VEL
LIN {X 0,Y 425.699,Z 281.752,A -85,B 0,C 180,E1 -9900,E2 -9900} C_VEL
LIN {X 0,Y 425.544,Z 281.781,A -85,B 0,C 180,E1 -9902.84,E2 -9902.84} C_VEL
LIN {X 0,Y 425.526,Z 281.782,A -85,B 0,C 180,E1 -9906.639,E2 -9906.639} C_VEL
LIN {X 0,Y 425.399,Z 281.797,A -85,B 0,C 180,E1 -9909.51,E2 -9909.51} C_VEL
LIN {X 0,Y 425.391,Z 281.806,A -85,B 0,C 180,E1 -9912.904,E2 -9912.904} C_VEL
LIN {X 0,Y 425.36,Z 281.799,A -85,B 0,C 180,E1 -9916.605,E2 -9916.605} C_VEL
LIN {X 0,Y 425.327,Z 281.812,A -85,B 0,C 180,E1 -9919.636,E2 -9919.636} C_VEL
LIN {X 0,Y 425.305,Z 281.814,A -85,B 0,C 180,E1 -9923.365,E2 -9923.365} C_VEL
LIN {X 0,Y 425.345,Z 281.803,A -85,B 0,C 180,E1 -9926.844,E2 -9926.844} C_VEL
LIN {X 0,Y 425.289,Z 281.818,A -85,B 0,C 180,E1 -9929.72,E2 -9929.72} C_VEL
LIN {X 0,Y 425.281,Z 281.824,A -85,B 0,C 180,E1 -9933.048,E2 -9933.048} C_VEL
LIN {X 0,Y 425.282,Z 281.819,A -85,B 0,C 180,E1 -9935.929,E2 -9935.929} C_VEL
LIN {X 0,Y 425.286,Z 281.813,A -85,B 0,C 180,E1 -9939.042,E2 -9939.042} C_VEL
LIN {X 0,Y 425.289,Z 281.81,A -85,B 0,C 180,E1 -9941.958,E2 -9941.958} C_VEL
LIN {X 0,Y 425.284,Z 281.814,A -85,B 0,C 180,E1 -9945.283,E2 -9945.283} C_VEL
LIN {X 0,Y 425.274,Z 281.825,A -85,B 0,C 180,E1 -9948.622,E2 -9948.622} C_VEL
LIN {X 0,Y 425.309,Z 281.815,A -85,B 0,C 180,E1 -9951.103,E2 -9951.103} C_VEL
LIN {X 0,Y 425.299,Z 281.82,A -85,B 0,C 180,E1 -9954.664,E2 -9954.664} C_VEL
LIN {X 0,Y 425.324,Z 281.855,A -85,B 0,C 180,E1 -9956.425,E2 -9956.425} C_VEL
LIN {X 0,Y 427.086,Z 287.425,A -85,B 0,C 180,E1 -9957.355,E2 -9957.355} C_VEL
LIN {X 0,Y 437.41,Z 307.383,A -85,B 0,C 180,E1 -9958.603,E2 -9958.603} C_VEL
LIN {X 0,Y 443.105,Z 319.368,A -85,B 0,C 180,E1 -9959.277,E2 -9959.277} C_VEL
LIN {X 0,Y 439.807,Z 489.56,A -85,B 0,C 180,E1 -9962.17,E2 -9962.17} C_VEL
LIN {X 0,Y 439.087,Z 506.482,A -85,B 0,C 180,E1 -9962.602,E2 -9962.602} C_VEL
LIN {X 0,Y 438.226,Z 522.296,A -85,B 0,C 180,E1 -9963.189,E2 -9963.189} C_VEL
LIN {X 0,Y 437.019,Z 537.885,A -85,B 0,C 180,E1 -9963.945,E2 -9963.945} C_VEL
LIN {X 0,Y 436.448,Z 544.786,A -85,B 0,C 180,E1 -9964.352,E2 -9964.352} C_VEL
LIN {X 0,Y 435.374,Z 550.163,A -85,B 0,C 180,E1 -9964.645,E2 -9964.645} C_VEL
LIN {X 0,Y 431.936,Z 558.887,A -85,B 0,C 180,E1 -9965.078,E2 -9965.078} C_VEL
LIN {X 0,Y 428.429,Z 567.332,A -85,B 0,C 180,E1 -9965.582,E2 -9965.582} C_VEL
LIN {X 0,Y 427.258,Z 572.266,A -85,B 0,C 180,E1 -9965.984,E2 -9965.984} C_VEL
LIN {X 0,Y 425.499,Z 586.856,A -85,B 0,C 180,E1 -9967.417,E2 -9967.417} C_VEL
LIN {X 0,Y 423.938,Z 599.144,A -85,B 0,C 180,E1 -9968.865,E2 -9968.865} C_VEL
LIN {X 0,Y 422.372,Z 611.367,A -85,B 0,C 180,E1 -9970.562,E2 -9970.562} C_VEL
LIN {X 0,Y 421.125,Z 621.339,A -85,B 0,C 180,E1 -9972.186,E2 -9972.186} C_VEL
LIN {X 0,Y 419.997,Z 630.692,A -85,B 0,C 180,E1 -9973.972,E2 -9973.972} C_VEL
LIN {X 0,Y 419.013,Z 639.267,A -85,B 0,C 180,E1 -9975.924,E2 -9975.924} C_VEL
LIN {X 0,Y 418.302,Z 646.438,A -85,B 0,C 180,E1 -9977.877,E2 -9977.877} C_VEL
LIN {X 0,Y 417.722,Z 652.375,A -85,B 0,C 180,E1 -9979.825,E2 -9979.825} C_VEL
LIN {X 0,Y 417.366,Z 658.121,A -85,B 0,C 180,E1 -9982.258,E2 -9982.258} C_VEL
LIN {X 0,Y 417.196,Z 661.488,A -85,B 0,C 180,E1 -9984.199,E2 -9984.199} C_VEL
LIN {X 0,Y 417.033,Z 663.937,A -85,B 0,C 180,E1 -9986.135,E2 -9986.135} C_VEL
LIN {X 0,Y 417.074,Z 665.326,A -85,B 0,C 180,E1 -9988.069,E2 -9988.069} C_VEL
LIN {X 0,Y 417.001,Z 665.866,A -85,B 0,C 180,E1 -9990,E2 -9990} C_VEL
LIN {X 0,Y 417.073,Z 665.373,A -85,B 0,C 180,E1 -9991.931,E2 -9991.931} C_VEL
LIN {X 0,Y 417.032,Z 664.029,A -85,B 0,C 180,E1 -9993.865,E2 -9993.865} C_VEL
LIN {X 0,Y 417.261,Z 660.724,A -85,B 0,C 180,E1 -9996.411,E2 -9996.411} C_VEL
LIN {X 0,Y 417.491,Z 656.215,A -85,B 0,C 180,E1 -9998.714,E2 -9998.714} C_VEL
LIN {X 0,Y 417.792,Z 651.236,A -85,B 0,C 180,E1 -10000.663,E2 -10000.663} C_VEL
LIN {X 0,Y 418.396,Z 645.141,A -85,B 0,C 180,E1 -10002.613,E2 -10002.613} C_VEL
LIN {X 0,Y 419.309,Z 636.654,A -85,B 0,C 180,E1 -10004.809,E2 -10004.809} C_VEL
LIN {X 0,Y 420.418,Z 627.492,A -85,B 0,C 180,E1 -10006.76,E2 -10006.76} C_VEL
LIN {X 0,Y 421.537,Z 618.064,A -85,B 0,C 180,E1 -10008.468,E2 -10008.468} C_VEL
LIN {X 0,Y 422.937,Z 607.065,A -85,B 0,C 180,E1 -10010.17,E2 -10010.17} C_VEL
LIN {X 0,Y 424.383,Z 595.475,A -85,B 0,C 180,E1 -10011.69,E2 -10011.69} C_VEL
LIN {X 0,Y 425.993,Z 583.066,A -85,B 0,C 180,E1 -10013.068,E2 -10013.068} C_VEL
LIN {X 0,Y 427.586,Z 569.036,A -85,B 0,C 180,E1 -10014.391,E2 -10014.391} C_VEL
LIN {X 0,Y 429.085,Z 555.589,A -85,B 0,C 180,E1 -10015.45,E2 -10015.45} C_VEL
LIN {X 0,Y 430.423,Z 540.621,A -85,B 0,C 180,E1 -10016.419,E2 -10016.419} C_VEL
LIN {X 0,Y 431.725,Z 525.719,A -85,B 0,C 180,E1 -10017.182,E2 -10017.182} C_VEL
LIN {X 0,Y 432.641,Z 510.302,A -85,B 0,C 180,E1 -10017.808,E2 -10017.808} C_VEL
LIN {X 0,Y 433.393,Z 495.442,A -85,B 0,C 180,E1 -10018.238,E2 -10018.238} C_VEL
LIN {X 0,Y 434.053,Z 467.832,A -85,B 0,C 180,E1 -10018.752,E2 -10018.752} C_VEL
LIN {X 0,Y 437.013,Z 321.585,A -85,B 0,C 180,E1 -10021.259,E2 -10021.259} C_VEL
LIN {X 0,Y 427.532,Z 301.957,A -85,B 0,C 180,E1 -10022.421,E2 -10022.421} C_VEL
LIN {X 0,Y 419.781,Z 287.388,A -85,B 0,C 180,E1 -10023.4,E2 -10023.4} C_VEL
LIN {X 0,Y 418.264,Z 282.701,A -85,B 0,C 180,E1 -10024.256,E2 -10024.256} C_VEL
LIN {X 0,Y 418.238,Z 282.684,A -85,B 0,C 180,E1 -10027.224,E2 -10027.224} C_VEL
LIN {X 0,Y 418.243,Z 282.695,A -85,B 0,C 180,E1 -10029.682,E2 -10029.682} C_VEL
LIN {X 0,Y 418.229,Z 282.695,A -85,B 0,C 180,E1 -10032.321,E2 -10032.321} C_VEL
LIN {X 0,Y 418.234,Z 282.695,A -85,B 0,C 180,E1 -10035.108,E2 -10035.108} C_VEL
LIN {X 0,Y 418.238,Z 282.697,A -85,B 0,C 180,E1 -10037.767,E2 -10037.767} C_VEL
LIN {X 0,Y 418.247,Z 282.697,A -85,B 0,C 180,E1 -10040.62,E2 -10040.62} C_VEL
LIN {X 0,Y 418.242,Z 282.696,A -85,B 0,C 180,E1 -10043.976,E2 -10043.976} C_VEL
LIN {X 0,Y 418.255,Z 282.687,A -85,B 0,C 180,E1 -10047.156,E2 -10047.156} C_VEL
LIN {X 0,Y 418.266,Z 282.694,A -85,B 0,C 180,E1 -10050.895,E2 -10050.895} C_VEL
LIN {X 0,Y 418.268,Z 282.692,A -85,B 0,C 180,E1 -10054.096,E2 -10054.096} C_VEL
LIN {X 0,Y 418.236,Z 282.685,A -85,B 0,C 180,E1 -10057.264,E2 -10057.264} C_VEL
LIN {X 0,Y 418.281,Z 282.692,A -85,B 0,C 180,E1 -10060.364,E2 -10060.364} C_VEL
LIN {X 0,Y 418.314,Z 282.672,A -85,B 0,C 180,E1 -10063.404,E2 -10063.404} C_VEL
LIN {X 0,Y 418.344,Z 282.689,A -85,B 0,C 180,E1 -10066.999,E2 -10066.999} C_VEL
LIN {X 0,Y 418.337,Z 282.667,A -85,B 0,C 180,E1 -10070.328,E2 -10070.328} C_VEL
LIN {X 0,Y 418.511,Z 282.658,A -85,B 0,C 180,E1 -10072.279,E2 -10072.279} C_VEL
LIN {X 0,Y 418.512,Z 282.664,A -85,B 0,C 180,E1 -10074.217,E2 -10074.217} C_VEL
LIN {X 0,Y 418.54,Z 282.647,A -85,B 0,C 180,E1 -10078.075,E2 -10078.075} C_VEL
LIN {X 0,Y 418.67,Z 282.643,A -85,B 0,C 180,E1 -10080,E2 -10080} C_VEL
LIN {X 0,Y 418.507,Z 282.652,A -85,B 0,C 180,E1 -10082.888,E2 -10082.888} C_VEL
LIN {X 0,Y 418.492,Z 282.667,A -85,B 0,C 180,E1 -10086.751,E2 -10086.751} C_VEL
LIN {X 0,Y 418.338,Z 282.672,A -85,B 0,C 180,E1 -10089.671,E2 -10089.671} C_VEL
LIN {X 0,Y 418.343,Z 282.687,A -85,B 0,C 180,E1 -10093.001,E2 -10093.001} C_VEL
LIN {X 0,Y 418.31,Z 282.693,A -85,B 0,C 180,E1 -10096.735,E2 -10096.735} C_VEL
LIN {X 0,Y 418.268,Z 282.695,A -85,B 0,C 180,E1 -10099.79,E2 -10099.79} C_VEL
LIN {X 0,Y 418.235,Z 282.703,A -85,B 0,C 180,E1 -10102.736,E2 -10102.736} C_VEL
LIN {X 0,Y 418.268,Z 282.697,A -85,B 0,C 180,E1 -10105.904,E2 -10105.904} C_VEL
LIN {X 0,Y 418.262,Z 282.699,A -85,B 0,C 180,E1 -10109.162,E2 -10109.162} C_VEL
LIN {X 0,Y 418.254,Z 282.7,A -85,B 0,C 180,E1 -10112.844,E2 -10112.844} C_VEL
LIN {X 0,Y 418.246,Z 282.699,A -85,B 0,C 180,E1 -10116.239,E2 -10116.239} C_VEL
LIN {X 0,Y 418.246,Z 282.701,A -85,B 0,C 180,E1 -10119.682,E2 -10119.682} C_VEL
LIN {X 0,Y 418.227,Z 282.706,A -85,B 0,C 180,E1 -10122.321,E2 -10122.321} C_VEL
LIN {X 0,Y 418.237,Z 282.704,A -85,B 0,C 180,E1 -10125.109,E2 -10125.109} C_VEL
LIN {X 0,Y 418.24,Z 282.701,A -85,B 0,C 180,E1 -10127.767,E2 -10127.767} C_VEL
LIN {X 0,Y 418.256,Z 282.701,A -85,B 0,C 180,E1 -10130.619,E2 -10130.619} C_VEL
